// Mitsubishi GX Works2 project: PLC   PLC: FX3G
// LABEL_TEST

// global labels: Global1
VAR_GLOBAL
  MODBUS AT M50 : BOOL;  (* Modbus ON/OFF *)
  WeatherPrognose AT M30 : BOOL;  (* Waether prognose download *)
  Nordpool : BOOL;  (* Nordpool price *)
  Manual : BOOL;  (* Manual price *)
  UP_15_00 : BOOL;  (* Nordpool/naual data update *)
  Ready AT M1 : BOOL;  (* Machine ready *)
  NordPtoGeraph AT M64 : BOOL;  (* Nordpool Prise to graph *)
  CopyDataToGraph : BOOL;  (* Manual/Nordpool data copyng to graph *)
  CopyDataToGraphIsReady : BOOL;  (* Prise data is copyed to graph *)
  SortDataReady : BOOL;  (* Start sort data prodsedure ready *)
  EnergyUseGraph : BOOL;  (* Effective energy use next 24h *)
  DataLoading : BOOL;  (* Data Loading flag *)
  SortDataStart : BOOL;  (* Start data sorting *)
  SortData : BOOL;  (* Start sort data prodsedure *)
  MoveData : BOOL;  (* Move data to sort register *)
  SortDataOK : BOOL;  (* Data is sorted *)
  MoveDataOK : BOOL;  (* Data is moved *)
  Sort24hHighMinOK : BOOL;  (* Data is sorted *)
  Sort24hMinHighOK : BOOL;  (* Data sorted *)
  Sort24hMinHigh24OK : BOOL;  (* Data sorted *)
  Sort24hMinHigh : BOOL;  (* Sort 24h prise min to hight *)
  Sort24hHighMin : BOOL;  (* Sort 24h prise hight to min *)
  Sort24hMinHigh24 : BOOL;  (* Sort 24h prise Min to High *)
  price : BOOL;  (* Add nordpool manual pice *)
  FindPriseMax : BOOL;  (* Find max value in graph *)
  FindPriseMaxOK : BOOL;  (* Find max value is ready *)
  WeatherNextDay : BOOL;  (* Start weather next day prognisis calc *)
  NextDayAvrTemp AT D1850 : DINT;  (* Next day prognosis temp *)
  NextDayAvrWind AT D1852 : DINT;  (* Next day prognosis wind *)
  NextDayAvrCloudy AT D1854 : DINT;  (* Next day avareage cloudy prognosis *)
  WeatherNextDayOK : BOOL;  (* Weather next day OK *)
  ReadEnergyRequirement : BOOL;  (* Read energy requirement form enegry table *)
  ReadEnergyWind : INT;  (* wind prognosis information *)
  ReadEnergyRadiation : INT;  (* Enegri inoramatsion from prognaosis *)
  EnergyDataFromTable : INT;  (* energy information from the data table *)
  WriteEnergyRequirement : BOOL;  (* Write erengy requirements to data table *)
  WriteEnergyWind : INT;  (* Write energy to data table *)
  EnergyDataFromLast24h : INT;  (* Energy data from Last24H *)
  priceOK : BOOL;  (* Prse is selected *)
  GraphicDataUpdate : BOOL;  (* Update graphics data *)
  GraphicDataUpdateOK : BOOL;  (* Graphics data is updated *)
  SortDataGrReady : BOOL;  (* Data sorted for graphics *)
  EnernyUseReady : BOOL;  (* Egery graph is updated *)
  CalcUsablePriceThreshold : BOOL;  (* Calculate usable (low price) price threshold *)
  PorgnosGetButton AT M36 : BOOL;  (* Prognose Button HMI *)
  ReadEnergyRequirementOK : BOOL;  (* Read energy requirement is readed *)
  WriteEnergyRequirementOK : BOOL;  (* Write energy requirement is writed *)
  HeatFlowLiters AT D68 : INT;  (* Heat flow l/min *)
  Wifi_SSID AT D200 : ARRAY [0..31] OF INT;  (* WIfi SSID name *)
  RadiatorHeatingPump : BOOL;  (* Radiator Heat Pump ON/Off *)
  FloorHeatingPump : BOOL;  (* Floor heating pump ON/Off *)
  HeaterHeatingPump : BOOL;  (* Heter heating pump ON/Off *)
  ElectricHeaterCenter : BOOL;  (* Electric heater center positsion ON/OFF *)
  ElectricHeaterLower AT M14 : BOOL;  (* Electric heater lower ON/OFF *)
  RadiatorHeatingActuatorState : INT;  (* Radiator valve actuator positsion (0-100%hot) *)
  OutsideTemp AT D56 : INT;  (* Outside temp x10 *)
  Ring1TargetTemp AT D58 : DINT;  (* Ring 1 (Radiator) Target Temp *)
  Ring2TargetTemp AT D70 : INT;  (* Target temerature for floor heating *)
  RadiatorHeatTemp AT D36 : DINT;  (* Radiator heating temperatuse to heat *)
  Ring1ValvePos : INT;  (* Ring 1 Valve positsion *)
  FloorHeatTemp AT D40 : INT;  (* Floof heating temperatuse to heat *)
  FloorHeatingActuatorState : INT;  (* Floor heating positsion state (0..100% hot) *)
  HeatingMode : BOOL;  (* Heating or summer mode *)
  ElectricHeatON AT M40 : BOOL;  (* Electric heat method is ON *)
  SolidHeatON AT M41 : BOOL;  (* Solid fuel heteing method is ON *)
  HeatPumpHeatingON AT M42 : BOOL;  (* Heating pump heteing method is ON *)
  ElectricElementON : BOOL;  (* Switch electric heat ON *)
  PriceNow AT D2004 : INT;  (* Energy price now *)
  ElectricElementON_Sol_Heat : BOOL;  (* Heat element Solid Heat func *)
  ElectricElementON_El_Heat : BOOL;  (* Heat element ON Electric Heat func. *)
  TankWaterCapacity AT D2006 : INT;  (* Tenk water capasity *)
  TankEnergyCapacity100 AT D72 : DINT;  (* Tank Energy Capacity 100 *)
  EnergyConsumption24h AT D2008 : DINT;  (* Energy consumption last 24h *)
  HetedEnergyInLastH AT D2012 : INT;  (* Heting energy in last hours *)
  EnergyConsumptionYesterday AT D2010 : DINT;  (* Energy consumption yesterday *)
  ElElementPower AT D2014 : INT;  (* Heting element power W *)
  HeatingReallTime AT D2020 : DINT;  (* Real time heating (W) *)
  HeatingArea AT D1874 : DINT;  (* Heating area (building areme m2) *)
  PreviousDayWind : INT;  (* Previous day wind prognosis *)
  PreviousDayTemp : INT;  (* Previous day temperature probnosis *)
  PreviousDayCloudy : INT;  (* Previous day cloudy prognosis *)
  SolarRadiationDayMax : INT;  (* Solar radiation max per day *)
  EnConsumptionPer_C : DINT;  (* Energy consumption per degree *)
END_VAR

PROGRAM MAIN
VAR
  GraphicDataProtsess : INT;  (* Graphic data protsess count *)
END_VAR
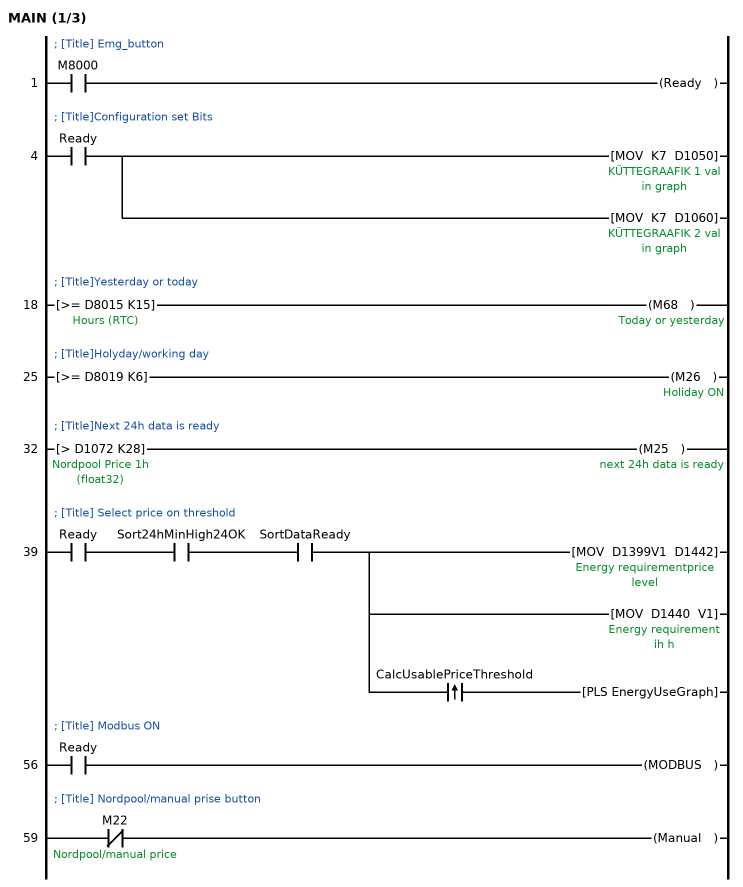
; [Title] Emg_button
1     LD      M8000
      OUT     Ready
; [Title]Configuration set Bits
4     LD      Ready
      MOV     K7 D1050  ; KÜTTEGRAAFIK 1 val in graph
        [note] 7 val. in heat cruve graph
      MOV     K7 D1060  ; KÜTTEGRAAFIK 2 val in graph
        [note] 7 val. in heat cruve graph
; [Title]Yesterday or today
18    LD>=    D8015 K15  ; Hours (RTC)
      OUT     M68  ; Today or yesterday
; [Title]Holyday/working day
25    LD>=    D8019 K6
      OUT     M26  ; Holiday ON
; [Title]Next 24h data is ready
32    LD>     D1072 K28  ; Nordpool Price 1h (float32)
      OUT     M25  ; next 24h data is ready
; [Title] Select price on threshold
39    LD      Ready
      AND     Sort24hMinHigh24OK
      AND     SortDataReady
      MOV     D1399V1 D1442  ; Energy requirementprice level
      MOV     D1440 V1  ; Energy requirement ih h
      ANDP    CalcUsablePriceThreshold
      PLS     EnergyUseGraph
; [Title] Modbus ON
56    LD      Ready
      OUT     MODBUS
; [Title] Nordpool/manual prise button
59    LDI     M22  ; Nordpool/manual price
      OUT     Manual
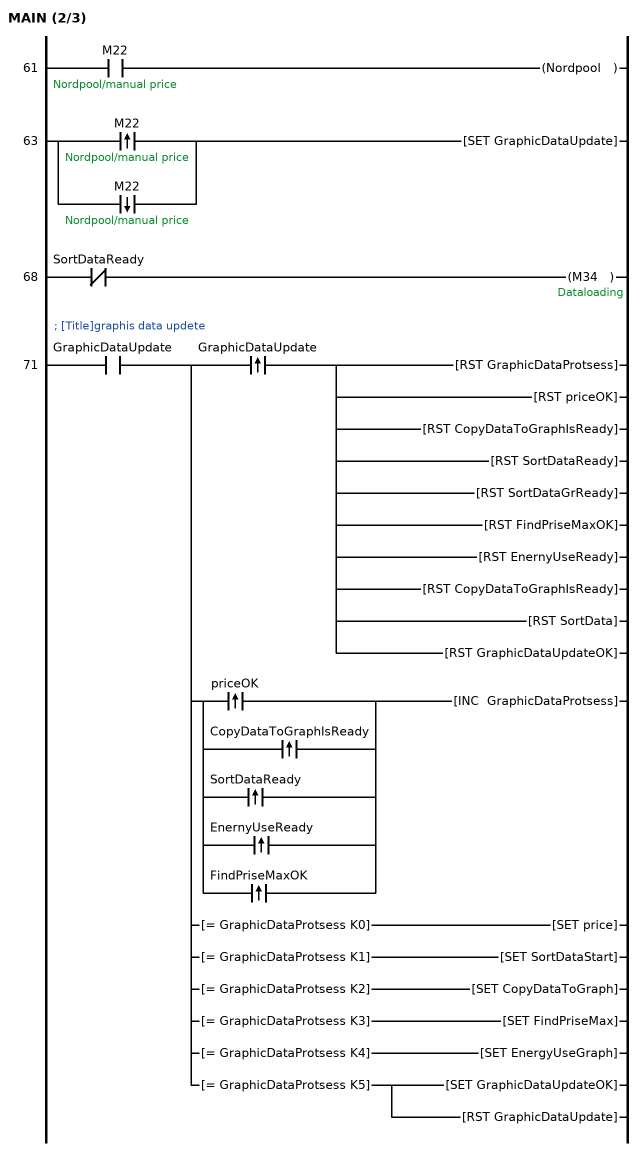
61    LD      M22  ; Nordpool/manual price
      OUT     Nordpool
63    LDP     M22  ; Nordpool/manual price
      ORF     M22  ; Nordpool/manual price
      SET     GraphicDataUpdate
68    LDI     SortDataReady
      OUT     M34  ; Dataloading
; [Title]graphis data updete
71    LD      GraphicDataUpdate
      MPS
      ANDP    GraphicDataUpdate
      RST     GraphicDataProtsess
      RST     priceOK
      RST     CopyDataToGraphIsReady
      RST     SortDataReady
      RST     SortDataGrReady
      RST     FindPriseMaxOK
      RST     EnernyUseReady
      RST     CopyDataToGraphIsReady
      RST     SortData
      RST     GraphicDataUpdateOK
      MRD
      LDP     priceOK
      ORP     CopyDataToGraphIsReady
      ORP     SortDataReady
      ORP     EnernyUseReady
      ORP     FindPriseMaxOK
      ANB
      INC     GraphicDataProtsess
      MRD
      AND=    GraphicDataProtsess K0
      SET     price
      MRD
      AND=    GraphicDataProtsess K1
      SET     SortDataStart
      MRD
      AND=    GraphicDataProtsess K2
      SET     CopyDataToGraph
      MRD
      AND=    GraphicDataProtsess K3
      SET     FindPriseMax
      MRD
      AND=    GraphicDataProtsess K4
      SET     EnergyUseGraph
      MPP
      AND=    GraphicDataProtsess K5
      SET     GraphicDataUpdateOK
      RST     GraphicDataUpdate
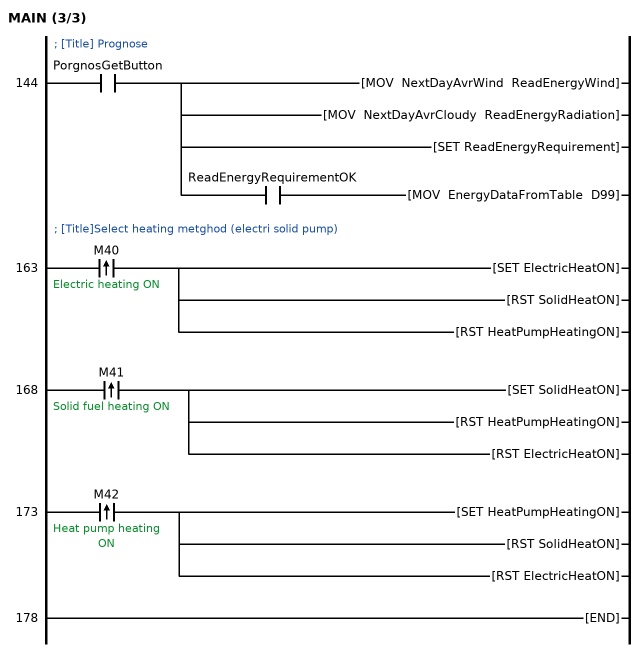
; [Title] Prognose
144   LD      PorgnosGetButton
      MOV     NextDayAvrWind ReadEnergyWind
      MOV     NextDayAvrCloudy ReadEnergyRadiation
      SET     ReadEnergyRequirement
      AND     ReadEnergyRequirementOK
      MOV     EnergyDataFromTable D99
; [Title]Select heating metghod (electri solid pump)
163   LDP     M40  ; Electric heating ON
      SET     ElectricHeatON
      RST     SolidHeatON
      RST     HeatPumpHeatingON
168   LDP     M41  ; Solid fuel heating ON
      SET     SolidHeatON
      RST     HeatPumpHeatingON
      RST     ElectricHeatON
173   LDP     M42  ; Heat pump heating ON
      SET     HeatPumpHeatingON
      RST     SolidHeatON
      RST     ElectricHeatON
178   END
END_PROGRAM

PROGRAM MODBUS
VAR
  ModBus_bnr : COUNTER;  (* Modbus comunicatsion block nr *)
  zxcv : BOOL;
END_VAR
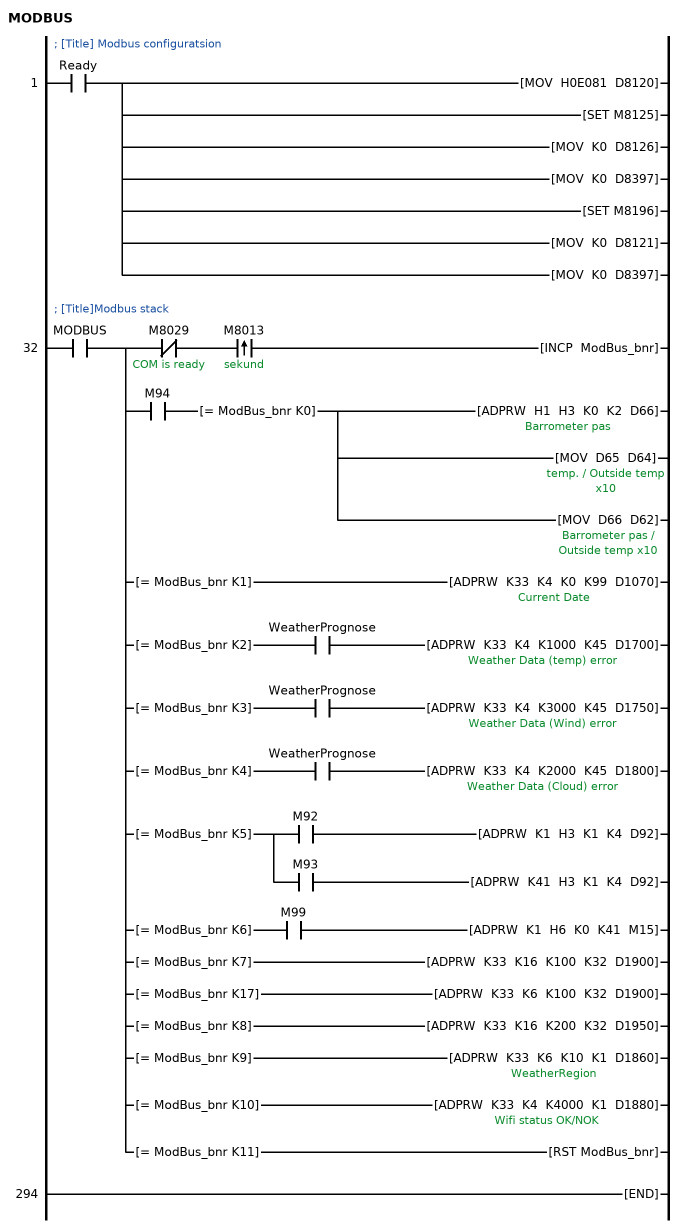
; [Title] Modbus configuratsion
1     LD      Ready
      MOV     H0E081 D8120
      SET     M8125
      MOV     K0 D8126
      MOV     K0 D8397
      SET     M8196
      MOV     K0 D8121
      MOV     K0 D8397
; [Title]Modbus stack
32    LD      MODBUS
      MPS
      ANI     M8029  ; COM is ready
      ANDP    M8013  ; sekund
      INCP    ModBus_bnr
        [note] barometer info
      MRD
      AND     M94
      AND=    ModBus_bnr K0
      ADPRW   H1 H3 K0 K2 D66  ; Barrometer pas
      MOV     D65 D64  ; temp. / Outside temp x10
      MOV     D66 D62  ; Outside temp x10
      MRD
      AND=    ModBus_bnr K1
      ADPRW   K33 K4 K0 K99 D1070  ; Current Date
        [note] Nordpool Data
      MRD
      AND=    ModBus_bnr K2
      AND     WeatherPrognose
      ADPRW   K33 K4 K1000 K45 D1700  ; Weather Data (temp) error
        [note] Weather Data (temp)
      MRD
      AND=    ModBus_bnr K3
      AND     WeatherPrognose
      ADPRW   K33 K4 K3000 K45 D1750  ; Weather Data (Wind) error
        [note] Weather Data (wind)
      MRD
      AND=    ModBus_bnr K4
      AND     WeatherPrognose
      ADPRW   K33 K4 K2000 K45 D1800  ; Weather Data (Cloud) error
        [note] Weather Data (cloudy%)
      MRD
      AND=    ModBus_bnr K5
      MPS
      AND     M92
      ADPRW   K1 H3 K1 K4 D92
        [note] Read pressure Data
      MPP
      AND     M93
      ADPRW   K41 H3 K1 K4 D92
        [note] Read pressure Data
      MRD
      AND=    ModBus_bnr K6
      AND     M99
      ADPRW   K1 H6 K0 K41 M15
        [note] PRESSURE SENSOR write MB 41
      MRD
      AND=    ModBus_bnr K7
      ADPRW   K33 K16 K100 K32 D1900
        [note] Wifi SSID
      MRD
      AND=    ModBus_bnr K17
      ADPRW   K33 K6 K100 K32 D1900
        [note] Wifi SSID
      MRD
      AND=    ModBus_bnr K8
      ADPRW   K33 K16 K200 K32 D1950
        [note] Wifi password
      MRD
      AND=    ModBus_bnr K9
      ADPRW   K33 K6 K10 K1 D1860  ; WeatherRegion
        [note] Weather region/loctsion
      MRD
      AND=    ModBus_bnr K10
      ADPRW   K33 K4 K4000 K1 D1880  ; Wifi status OK/NOK
        [note] Weather region/loctsion
      MPP
      AND=    ModBus_bnr K11
      RST     ModBus_bnr
294   END
END_PROGRAM

PROGRAM PRICE
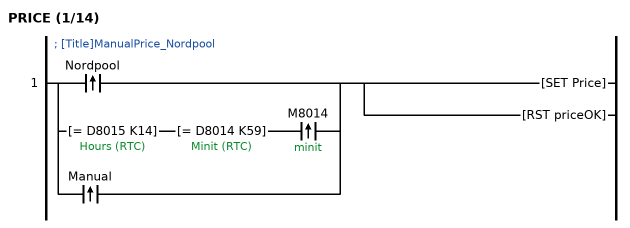
; [Title]ManualPrice_Nordpool
1     LDP     Nordpool
      LD=     D8015 K14  ; Hours (RTC)
      AND=    D8014 K59  ; Minit (RTC)
      ANDP    M8014  ; minit
      ORB
      ORP     Manual
      SET     Price
      RST     priceOK
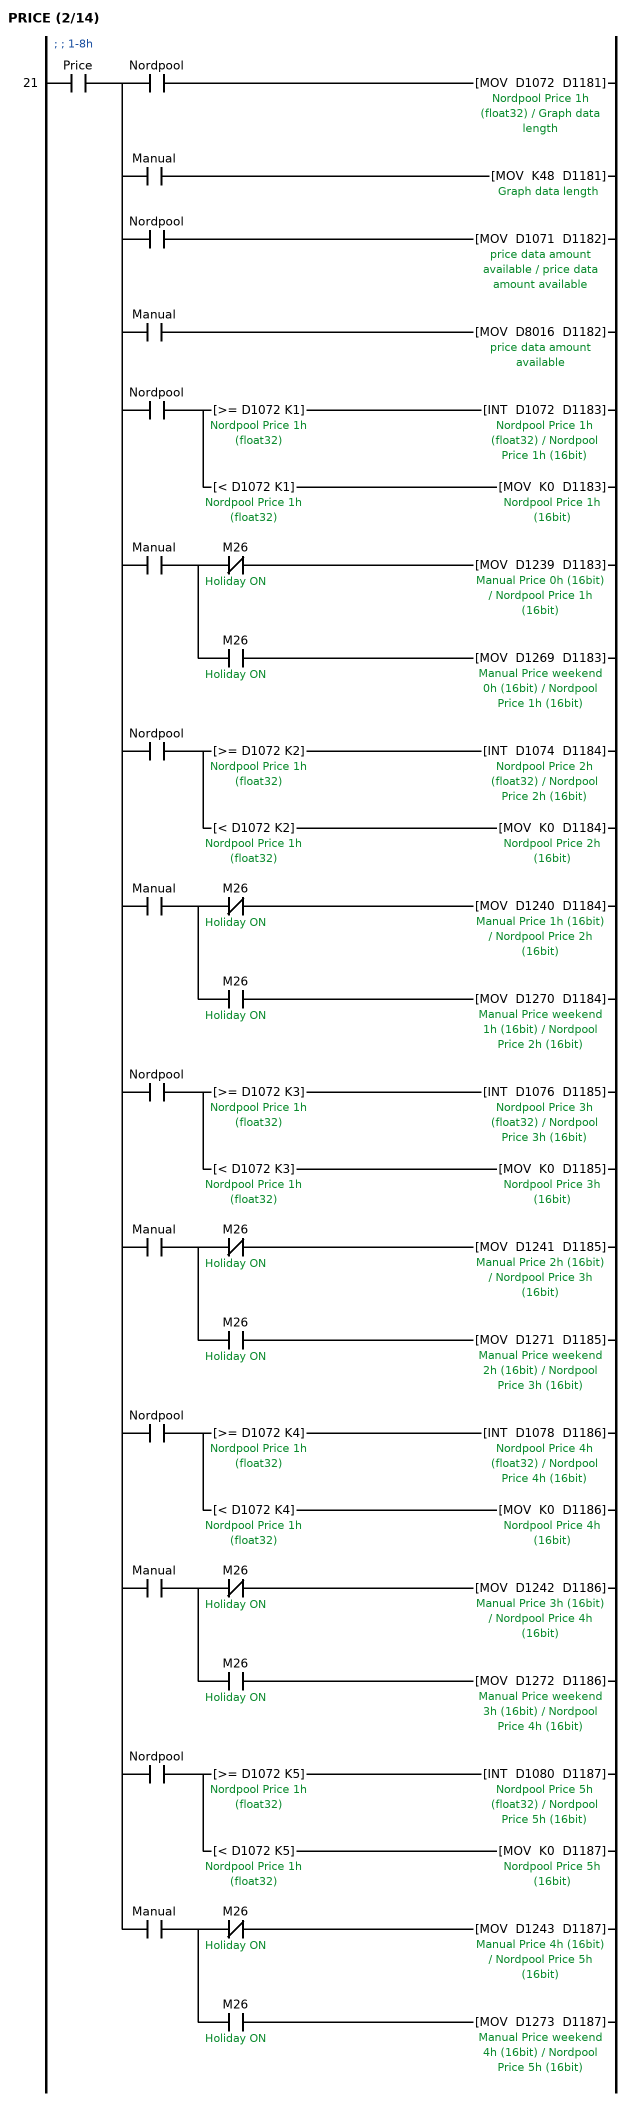
;  1-8h
21    LD      Price
      MPS
      AND     Nordpool
      MOV     D1072 D1181  ; Nordpool Price 1h (float32) / Graph data length
        [note] 00-01
      MRD
      AND     Manual
      MOV     K48 D1181
      MRD
      AND     Nordpool
      MOV     D1071 D1182  ; price data amount available / price data amount available
      MRD
      AND     Manual
      MOV     D8016 D1182
      MRD
      AND     Nordpool
      MPS
      AND>=   D1072 K1  ; Nordpool Price 1h (float32)
      INT     D1072 D1183  ; Nordpool Price 1h (16bit)
      MPP
      AND<    D1072 K1  ; Nordpool Price 1h (float32)
      MOV     K0 D1183
      MRD
      AND     Manual
      MPS
      ANI     M26  ; Holiday ON
      MOV     D1239 D1183  ; Manual Price 0h (16bit)
      MPP
      AND     M26  ; Holiday ON
      MOV     D1269 D1183  ; Manual Price weekend 0h (16bit)
      MRD
      AND     Nordpool
      MPS
      AND>=   D1072 K2  ; Nordpool Price 1h (float32)
      INT     D1074 D1184  ; Nordpool Price 2h (float32) / Nordpool Price 2h (16bit)
        [note] 01-02
      MPP
      AND<    D1072 K2  ; Nordpool Price 1h (float32)
      MOV     K0 D1184
      MRD
      AND     Manual
      MPS
      ANI     M26  ; Holiday ON
      MOV     D1240 D1184  ; Manual Price 1h (16bit)
      MPP
      AND     M26  ; Holiday ON
      MOV     D1270 D1184  ; Manual Price weekend 1h (16bit)
      MRD
      AND     Nordpool
      MPS
      AND>=   D1072 K3  ; Nordpool Price 1h (float32)
      INT     D1076 D1185  ; Nordpool Price 3h (float32) / Nordpool Price 3h (16bit)
        [note] 02-03
      MPP
      AND<    D1072 K3  ; Nordpool Price 1h (float32)
      MOV     K0 D1185
      MRD
      AND     Manual
      MPS
      ANI     M26  ; Holiday ON
      MOV     D1241 D1185  ; Manual Price 2h (16bit)
      MPP
      AND     M26  ; Holiday ON
      MOV     D1271 D1185  ; Manual Price weekend 2h (16bit)
      MRD
      AND     Nordpool
      MPS
      AND>=   D1072 K4  ; Nordpool Price 1h (float32)
      INT     D1078 D1186  ; Nordpool Price 4h (float32) / Nordpool Price 4h (16bit)
        [note] 03-04
      MPP
      AND<    D1072 K4  ; Nordpool Price 1h (float32)
      MOV     K0 D1186
      MRD
      AND     Manual
      MPS
      ANI     M26  ; Holiday ON
      MOV     D1242 D1186  ; Manual Price 3h (16bit)
      MPP
      AND     M26  ; Holiday ON
      MOV     D1272 D1186  ; Manual Price weekend 3h (16bit)
      MRD
      AND     Nordpool
      MPS
      AND>=   D1072 K5  ; Nordpool Price 1h (float32)
      INT     D1080 D1187  ; Nordpool Price 5h (float32) / Nordpool Price 5h (16bit)
        [note] 04-05
      MPP
      AND<    D1072 K5  ; Nordpool Price 1h (float32)
      MOV     K0 D1187
      MPP
      AND     Manual
      MPS
      ANI     M26  ; Holiday ON
      MOV     D1243 D1187  ; Manual Price 4h (16bit)
      MPP
      AND     M26  ; Holiday ON
      MOV     D1273 D1187  ; Manual Price weekend 4h (16bit)
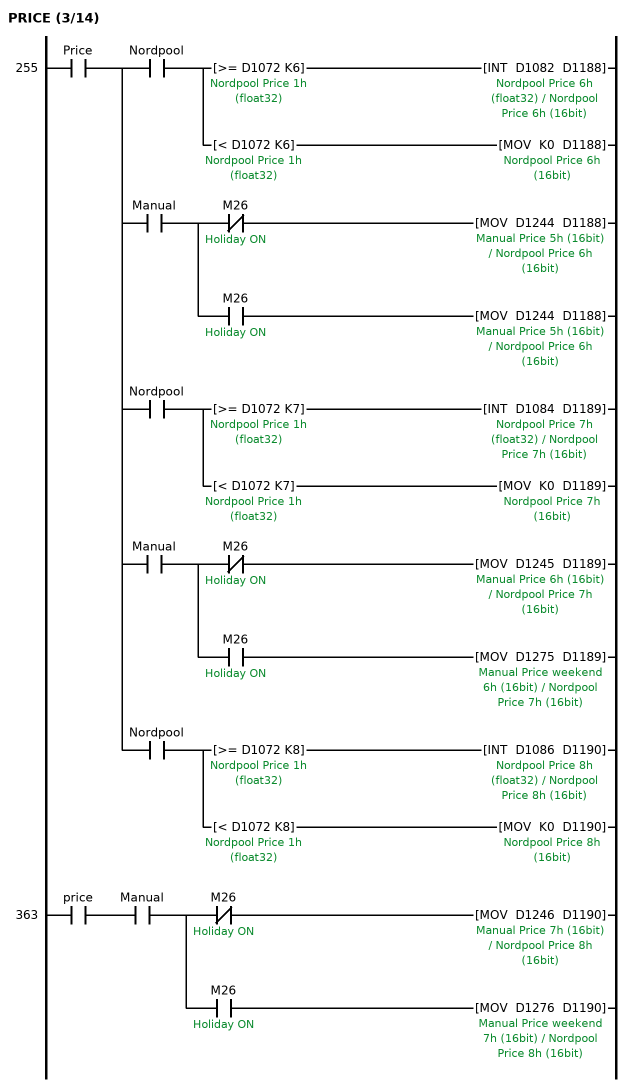
255   LD      Price
      MPS
      AND     Nordpool
      MPS
      AND>=   D1072 K6  ; Nordpool Price 1h (float32)
      INT     D1082 D1188  ; Nordpool Price 6h (float32) / Nordpool Price 6h (16bit)
        [note] 05-06
      MPP
      AND<    D1072 K6  ; Nordpool Price 1h (float32)
      MOV     K0 D1188
      MRD
      AND     Manual
      MPS
      ANI     M26  ; Holiday ON
      MOV     D1244 D1188  ; Manual Price 5h (16bit)
      MPP
      AND     M26  ; Holiday ON
      MOV     D1244 D1188
      MRD
      AND     Nordpool
      MPS
      AND>=   D1072 K7  ; Nordpool Price 1h (float32)
      INT     D1084 D1189  ; Nordpool Price 7h (float32) / Nordpool Price 7h (16bit)
        [note] 06-07
      MPP
      AND<    D1072 K7  ; Nordpool Price 1h (float32)
      MOV     K0 D1189
      MRD
      AND     Manual
      MPS
      ANI     M26  ; Holiday ON
      MOV     D1245 D1189  ; Manual Price 6h (16bit)
      MPP
      AND     M26  ; Holiday ON
      MOV     D1275 D1189  ; Manual Price weekend 6h (16bit)
      MPP
      AND     Nordpool
      MPS
      AND>=   D1072 K8  ; Nordpool Price 1h (float32)
      INT     D1086 D1190  ; Nordpool Price 8h (float32) / Nordpool Price 8h (16bit)
        [note] 07-08
      MPP
      AND<    D1072 K8  ; Nordpool Price 1h (float32)
      MOV     K0 D1190
363   LD      price
      AND     Manual
      MPS
      ANI     M26  ; Holiday ON
      MOV     D1246 D1190  ; Manual Price 7h (16bit)
      MPP
      AND     M26  ; Holiday ON
      MOV     D1276 D1190  ; Manual Price weekend 7h (16bit)
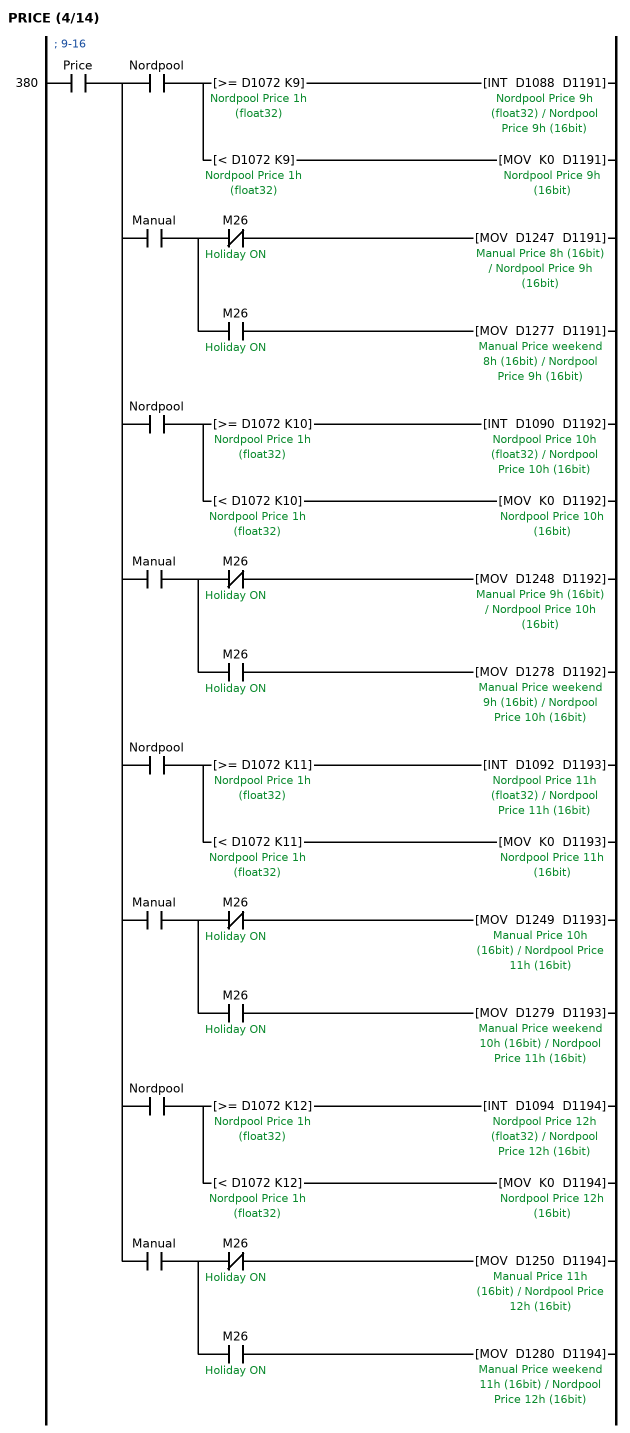
; 9-16
380   LD      Price
      MPS
      AND     Nordpool
      MPS
      AND>=   D1072 K9  ; Nordpool Price 1h (float32)
      INT     D1088 D1191  ; Nordpool Price 9h (float32) / Nordpool Price 9h (16bit)
        [note] 08-09
      MPP
      AND<    D1072 K9  ; Nordpool Price 1h (float32)
      MOV     K0 D1191
      MRD
      AND     Manual
      MPS
      ANI     M26  ; Holiday ON
      MOV     D1247 D1191  ; Manual Price 8h (16bit)
      MPP
      AND     M26  ; Holiday ON
      MOV     D1277 D1191  ; Manual Price weekend 8h (16bit)
      MRD
      AND     Nordpool
      MPS
      AND>=   D1072 K10  ; Nordpool Price 1h (float32)
      INT     D1090 D1192  ; Nordpool Price 10h (float32) / Nordpool Price 10h (16bit)
        [note] 9-10
      MPP
      AND<    D1072 K10  ; Nordpool Price 1h (float32)
      MOV     K0 D1192
      MRD
      AND     Manual
      MPS
      ANI     M26  ; Holiday ON
      MOV     D1248 D1192  ; Manual Price 9h (16bit)
      MPP
      AND     M26  ; Holiday ON
      MOV     D1278 D1192  ; Manual Price weekend 9h (16bit)
      MRD
      AND     Nordpool
      MPS
      AND>=   D1072 K11  ; Nordpool Price 1h (float32)
      INT     D1092 D1193  ; Nordpool Price 11h (float32) / Nordpool Price 11h (16bit)
        [note] 10-11
      MPP
      AND<    D1072 K11  ; Nordpool Price 1h (float32)
      MOV     K0 D1193
      MRD
      AND     Manual
      MPS
      ANI     M26  ; Holiday ON
      MOV     D1249 D1193  ; Manual Price 10h (16bit)
      MPP
      AND     M26  ; Holiday ON
      MOV     D1279 D1193  ; Manual Price weekend 10h (16bit)
      MRD
      AND     Nordpool
      MPS
      AND>=   D1072 K12  ; Nordpool Price 1h (float32)
      INT     D1094 D1194  ; Nordpool Price 12h (float32) / Nordpool Price 12h (16bit)
        [note] 11-12
      MPP
      AND<    D1072 K12  ; Nordpool Price 1h (float32)
      MOV     K0 D1194
      MPP
      AND     Manual
      MPS
      ANI     M26  ; Holiday ON
      MOV     D1250 D1194  ; Manual Price 11h (16bit)
      MPP
      AND     M26  ; Holiday ON
      MOV     D1280 D1194  ; Manual Price weekend 11h (16bit)
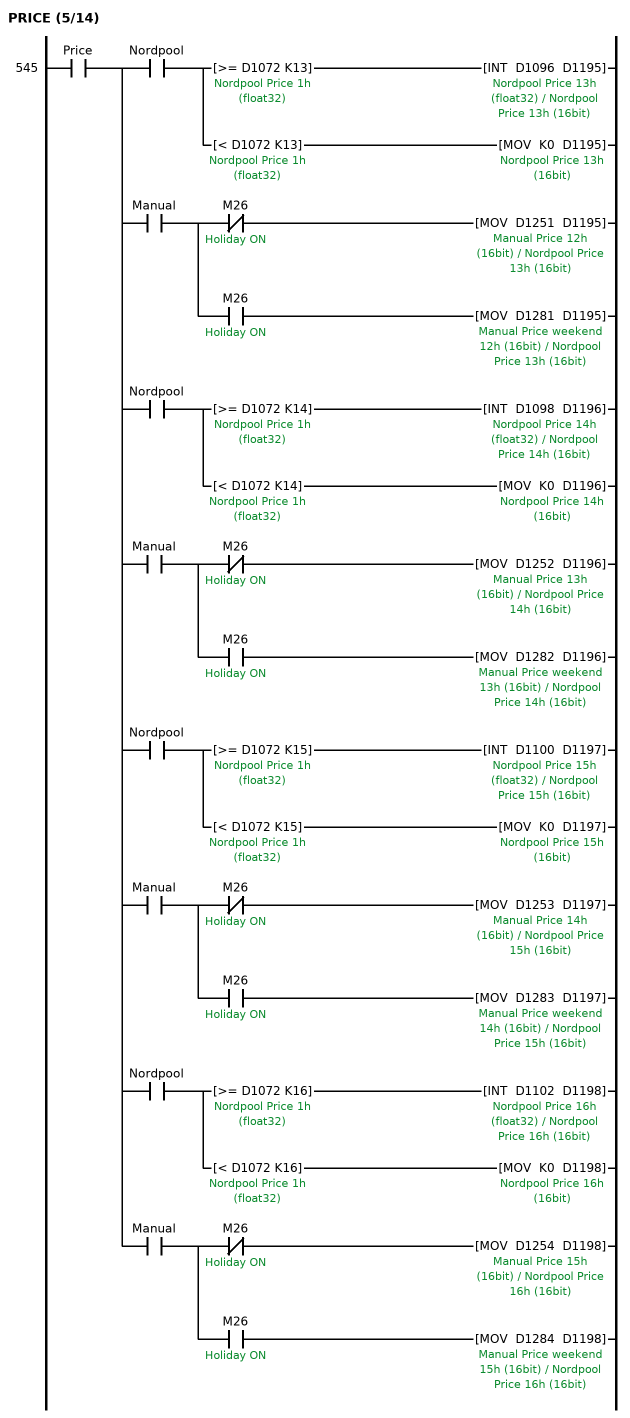
545   LD      Price
      MPS
      AND     Nordpool
      MPS
      AND>=   D1072 K13  ; Nordpool Price 1h (float32)
      INT     D1096 D1195  ; Nordpool Price 13h (float32) / Nordpool Price 13h (16bit)
        [note] 12-13
      MPP
      AND<    D1072 K13  ; Nordpool Price 1h (float32)
      MOV     K0 D1195
      MRD
      AND     Manual
      MPS
      ANI     M26  ; Holiday ON
      MOV     D1251 D1195  ; Manual Price 12h (16bit)
      MPP
      AND     M26  ; Holiday ON
      MOV     D1281 D1195  ; Manual Price weekend 12h (16bit)
      MRD
      AND     Nordpool
      MPS
      AND>=   D1072 K14  ; Nordpool Price 1h (float32)
      INT     D1098 D1196  ; Nordpool Price 14h (float32) / Nordpool Price 14h (16bit)
        [note] 13-14
      MPP
      AND<    D1072 K14  ; Nordpool Price 1h (float32)
      MOV     K0 D1196
      MRD
      AND     Manual
      MPS
      ANI     M26  ; Holiday ON
      MOV     D1252 D1196  ; Manual Price 13h (16bit)
      MPP
      AND     M26  ; Holiday ON
      MOV     D1282 D1196  ; Manual Price weekend 13h (16bit)
      MRD
      AND     Nordpool
      MPS
      AND>=   D1072 K15  ; Nordpool Price 1h (float32)
      INT     D1100 D1197  ; Nordpool Price 15h (float32) / Nordpool Price 15h (16bit)
        [note] 14-15
      MPP
      AND<    D1072 K15  ; Nordpool Price 1h (float32)
      MOV     K0 D1197
      MRD
      AND     Manual
      MPS
      ANI     M26  ; Holiday ON
      MOV     D1253 D1197  ; Manual Price 14h (16bit)
      MPP
      AND     M26  ; Holiday ON
      MOV     D1283 D1197  ; Manual Price weekend 14h (16bit)
      MRD
      AND     Nordpool
      MPS
      AND>=   D1072 K16  ; Nordpool Price 1h (float32)
      INT     D1102 D1198  ; Nordpool Price 16h (float32) / Nordpool Price 16h (16bit)
        [note] 15-16
      MPP
      AND<    D1072 K16  ; Nordpool Price 1h (float32)
      MOV     K0 D1198
      MPP
      AND     Manual
      MPS
      ANI     M26  ; Holiday ON
      MOV     D1254 D1198  ; Manual Price 15h (16bit)
      MPP
      AND     M26  ; Holiday ON
      MOV     D1284 D1198  ; Manual Price weekend 15h (16bit)
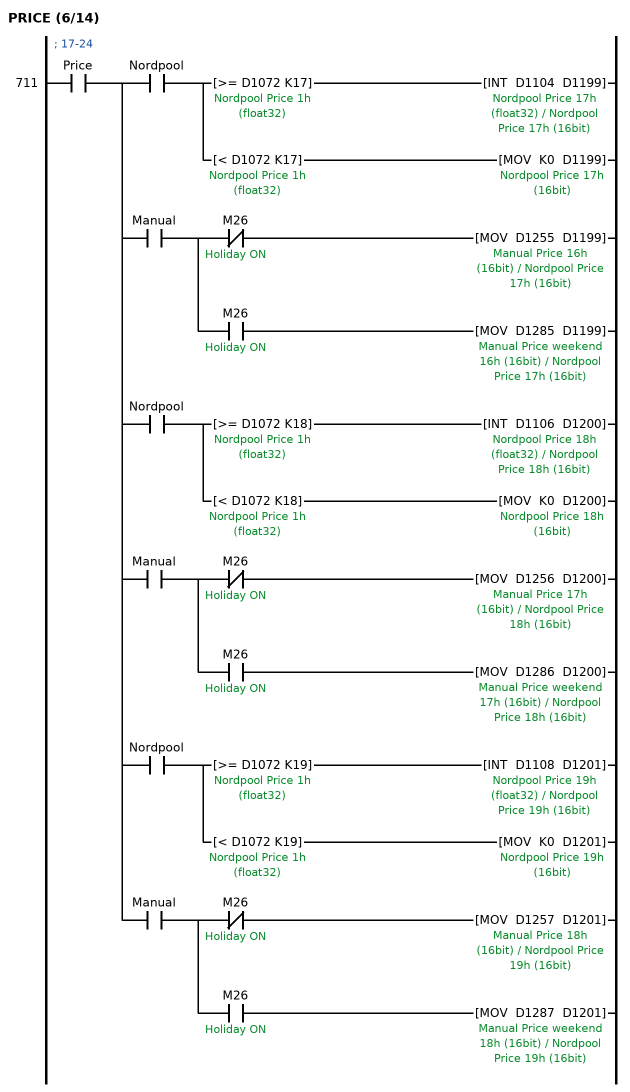
; 17-24
711   LD      Price
      MPS
      AND     Nordpool
      MPS
      AND>=   D1072 K17  ; Nordpool Price 1h (float32)
      INT     D1104 D1199  ; Nordpool Price 17h (float32) / Nordpool Price 17h (16bit)
        [note] 16-17
      MPP
      AND<    D1072 K17  ; Nordpool Price 1h (float32)
      MOV     K0 D1199
      MRD
      AND     Manual
      MPS
      ANI     M26  ; Holiday ON
      MOV     D1255 D1199  ; Manual Price 16h (16bit)
      MPP
      AND     M26  ; Holiday ON
      MOV     D1285 D1199  ; Manual Price weekend 16h (16bit)
      MRD
      AND     Nordpool
      MPS
      AND>=   D1072 K18  ; Nordpool Price 1h (float32)
      INT     D1106 D1200  ; Nordpool Price 18h (float32) / Nordpool Price 18h (16bit)
        [note] 17-18
      MPP
      AND<    D1072 K18  ; Nordpool Price 1h (float32)
      MOV     K0 D1200
      MRD
      AND     Manual
      MPS
      ANI     M26  ; Holiday ON
      MOV     D1256 D1200  ; Manual Price 17h (16bit)
      MPP
      AND     M26  ; Holiday ON
      MOV     D1286 D1200  ; Manual Price weekend 17h (16bit)
      MRD
      AND     Nordpool
      MPS
      AND>=   D1072 K19  ; Nordpool Price 1h (float32)
      INT     D1108 D1201  ; Nordpool Price 19h (float32) / Nordpool Price 19h (16bit)
        [note] 18-19
      MPP
      AND<    D1072 K19  ; Nordpool Price 1h (float32)
      MOV     K0 D1201
      MPP
      AND     Manual
      MPS
      ANI     M26  ; Holiday ON
      MOV     D1257 D1201  ; Manual Price 18h (16bit)
      MPP
      AND     M26  ; Holiday ON
      MOV     D1287 D1201  ; Manual Price weekend 18h (16bit)
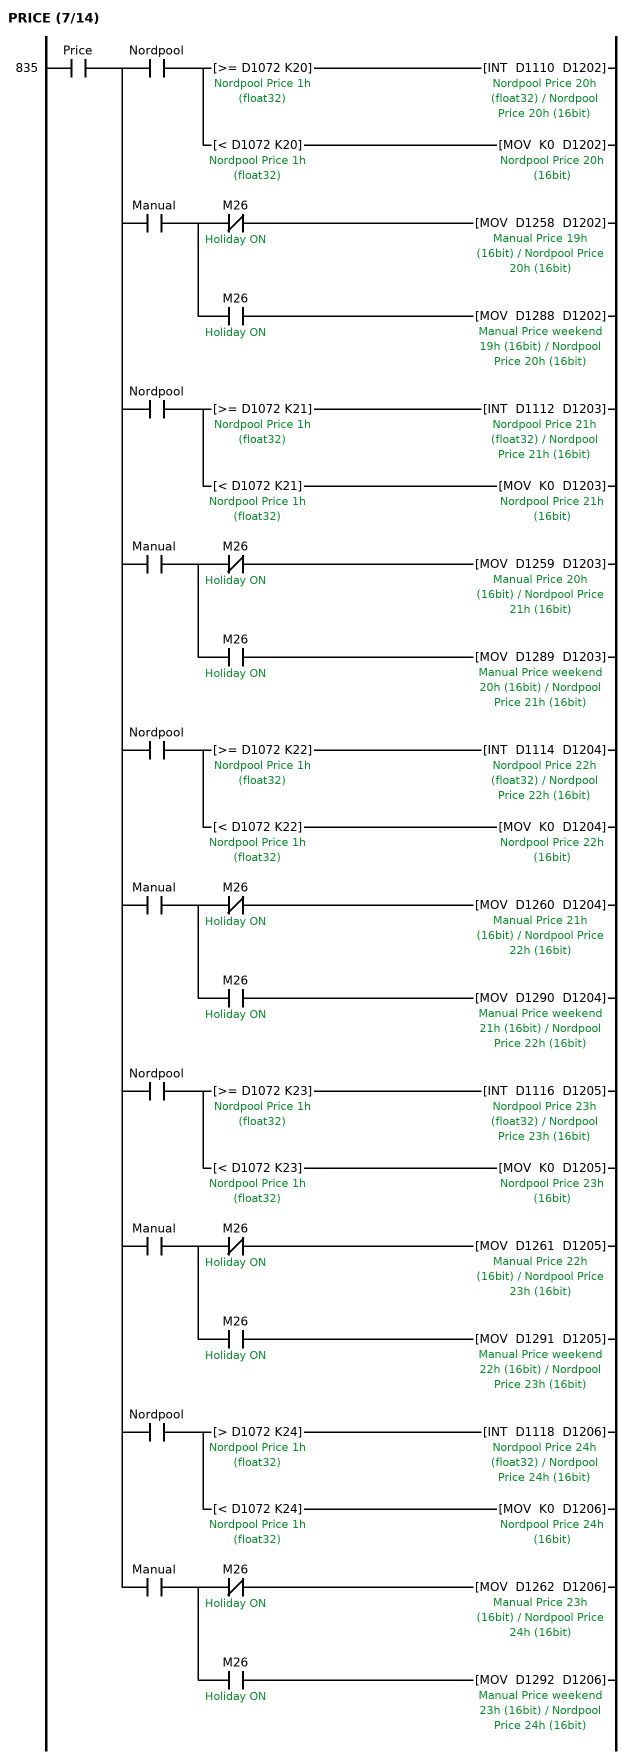
835   LD      Price
      MPS
      AND     Nordpool
      MPS
      AND>=   D1072 K20  ; Nordpool Price 1h (float32)
      INT     D1110 D1202  ; Nordpool Price 20h (float32) / Nordpool Price 20h (16bit)
        [note] 19-20
      MPP
      AND<    D1072 K20  ; Nordpool Price 1h (float32)
      MOV     K0 D1202
      MRD
      AND     Manual
      MPS
      ANI     M26  ; Holiday ON
      MOV     D1258 D1202  ; Manual Price 19h (16bit)
      MPP
      AND     M26  ; Holiday ON
      MOV     D1288 D1202  ; Manual Price weekend 19h (16bit)
      MRD
      AND     Nordpool
      MPS
      AND>=   D1072 K21  ; Nordpool Price 1h (float32)
      INT     D1112 D1203  ; Nordpool Price 21h (float32) / Nordpool Price 21h (16bit)
        [note] 20-21
      MPP
      AND<    D1072 K21  ; Nordpool Price 1h (float32)
      MOV     K0 D1203
      MRD
      AND     Manual
      MPS
      ANI     M26  ; Holiday ON
      MOV     D1259 D1203  ; Manual Price 20h (16bit)
      MPP
      AND     M26  ; Holiday ON
      MOV     D1289 D1203  ; Manual Price weekend 20h (16bit)
      MRD
      AND     Nordpool
      MPS
      AND>=   D1072 K22  ; Nordpool Price 1h (float32)
      INT     D1114 D1204  ; Nordpool Price 22h (float32) / Nordpool Price 22h (16bit)
        [note] 21-22
      MPP
      AND<    D1072 K22  ; Nordpool Price 1h (float32)
      MOV     K0 D1204
      MRD
      AND     Manual
      MPS
      ANI     M26  ; Holiday ON
      MOV     D1260 D1204  ; Manual Price 21h (16bit)
      MPP
      AND     M26  ; Holiday ON
      MOV     D1290 D1204  ; Manual Price weekend 21h (16bit)
      MRD
      AND     Nordpool
      MPS
      AND>=   D1072 K23  ; Nordpool Price 1h (float32)
      INT     D1116 D1205  ; Nordpool Price 23h (float32) / Nordpool Price 23h (16bit)
        [note] 22-23
      MPP
      AND<    D1072 K23  ; Nordpool Price 1h (float32)
      MOV     K0 D1205
      MRD
      AND     Manual
      MPS
      ANI     M26  ; Holiday ON
      MOV     D1261 D1205  ; Manual Price 22h (16bit)
      MPP
      AND     M26  ; Holiday ON
      MOV     D1291 D1205  ; Manual Price weekend 22h (16bit)
      MRD
      AND     Nordpool
      MPS
      AND>    D1072 K24  ; Nordpool Price 1h (float32)
      INT     D1118 D1206  ; Nordpool Price 24h (float32) / Nordpool Price 24h (16bit)
        [note] 23-00
      MPP
      AND<    D1072 K24  ; Nordpool Price 1h (float32)
      MOV     K0 D1206
      MPP
      AND     Manual
      MPS
      ANI     M26  ; Holiday ON
      MOV     D1262 D1206  ; Manual Price 23h (16bit)
      MPP
      AND     M26  ; Holiday ON
      MOV     D1292 D1206  ; Manual Price weekend 23h (16bit)
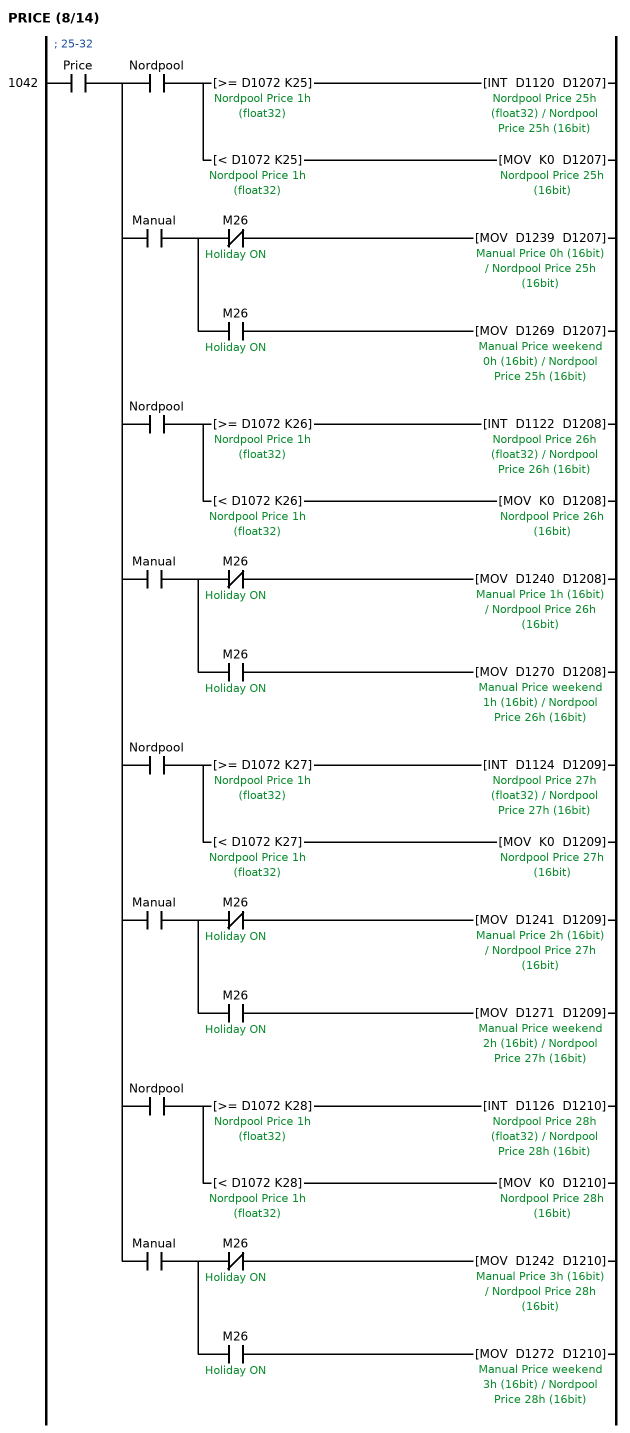
; 25-32
1042  LD      Price
      MPS
      AND     Nordpool
      MPS
      AND>=   D1072 K25  ; Nordpool Price 1h (float32)
      INT     D1120 D1207  ; Nordpool Price 25h (float32) / Nordpool Price 25h (16bit)
        [note] 25-26 (00-01)
      MPP
      AND<    D1072 K25  ; Nordpool Price 1h (float32)
      MOV     K0 D1207
      MRD
      AND     Manual
      MPS
      ANI     M26  ; Holiday ON
      MOV     D1239 D1207
      MPP
      AND     M26  ; Holiday ON
      MOV     D1269 D1207
      MRD
      AND     Nordpool
      MPS
      AND>=   D1072 K26  ; Nordpool Price 1h (float32)
      INT     D1122 D1208  ; Nordpool Price 26h (float32) / Nordpool Price 26h (16bit)
        [note] 26-27 (01-02)
      MPP
      AND<    D1072 K26  ; Nordpool Price 1h (float32)
      MOV     K0 D1208
      MRD
      AND     Manual
      MPS
      ANI     M26  ; Holiday ON
      MOV     D1240 D1208
      MPP
      AND     M26  ; Holiday ON
      MOV     D1270 D1208
      MRD
      AND     Nordpool
      MPS
      AND>=   D1072 K27  ; Nordpool Price 1h (float32)
      INT     D1124 D1209  ; Nordpool Price 27h (float32) / Nordpool Price 27h (16bit)
        [note] 27-28 (02-03)
      MPP
      AND<    D1072 K27  ; Nordpool Price 1h (float32)
      MOV     K0 D1209
      MRD
      AND     Manual
      MPS
      ANI     M26  ; Holiday ON
      MOV     D1241 D1209
      MPP
      AND     M26  ; Holiday ON
      MOV     D1271 D1209
      MRD
      AND     Nordpool
      MPS
      AND>=   D1072 K28  ; Nordpool Price 1h (float32)
      INT     D1126 D1210  ; Nordpool Price 28h (float32) / Nordpool Price 28h (16bit)
        [note] 28-29 (03-04)
      MPP
      AND<    D1072 K28  ; Nordpool Price 1h (float32)
      MOV     K0 D1210
      MPP
      AND     Manual
      MPS
      ANI     M26  ; Holiday ON
      MOV     D1242 D1210
      MPP
      AND     M26  ; Holiday ON
      MOV     D1272 D1210
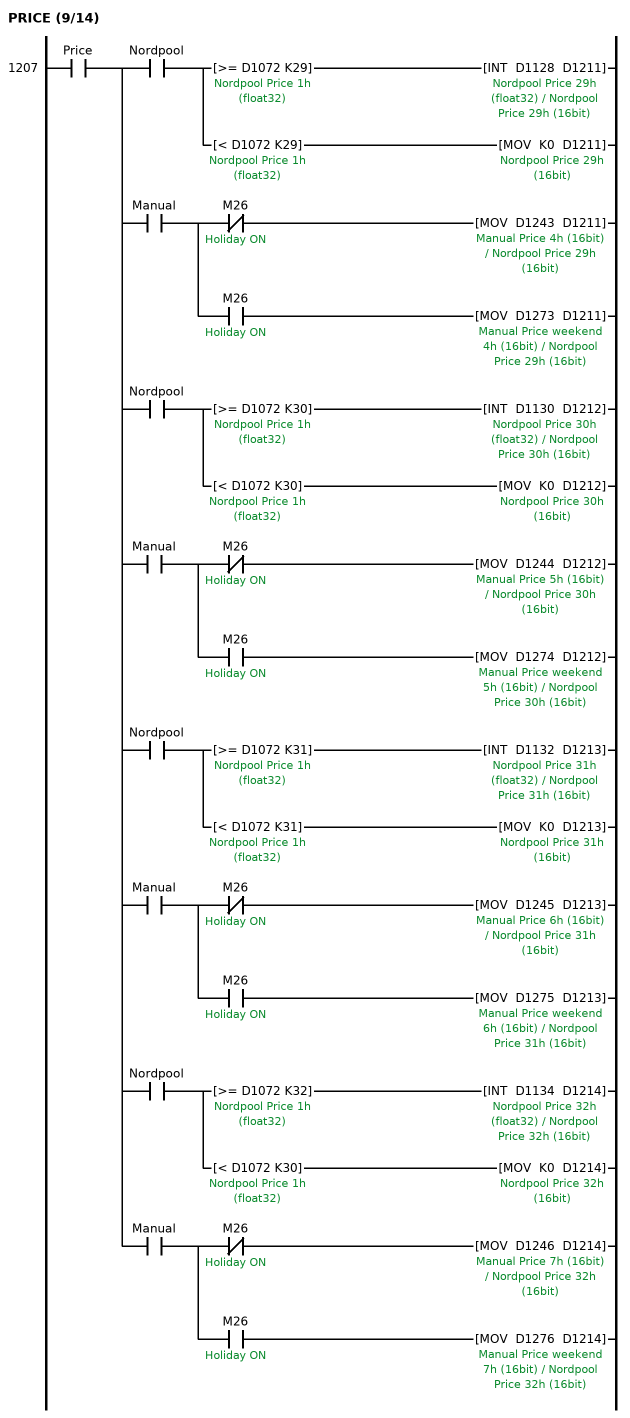
1207  LD      Price
      MPS
      AND     Nordpool
      MPS
      AND>=   D1072 K29  ; Nordpool Price 1h (float32)
      INT     D1128 D1211  ; Nordpool Price 29h (float32) / Nordpool Price 29h (16bit)
        [note] 29-30 (04-05)
      MPP
      AND<    D1072 K29  ; Nordpool Price 1h (float32)
      MOV     K0 D1211
      MRD
      AND     Manual
      MPS
      ANI     M26  ; Holiday ON
      MOV     D1243 D1211
      MPP
      AND     M26  ; Holiday ON
      MOV     D1273 D1211
      MRD
      AND     Nordpool
      MPS
      AND>=   D1072 K30  ; Nordpool Price 1h (float32)
      INT     D1130 D1212  ; Nordpool Price 30h (float32) / Nordpool Price 30h (16bit)
        [note] ; 30-31 (05-06)
      MPP
      AND<    D1072 K30  ; Nordpool Price 1h (float32)
      MOV     K0 D1212
      MRD
      AND     Manual
      MPS
      ANI     M26  ; Holiday ON
      MOV     D1244 D1212
      MPP
      AND     M26  ; Holiday ON
      MOV     D1274 D1212  ; Manual Price weekend 5h (16bit)
      MRD
      AND     Nordpool
      MPS
      AND>=   D1072 K31  ; Nordpool Price 1h (float32)
      INT     D1132 D1213  ; Nordpool Price 31h (float32) / Nordpool Price 31h (16bit)
        [note] 31-32 (06-07)
      MPP
      AND<    D1072 K31  ; Nordpool Price 1h (float32)
      MOV     K0 D1213
      MRD
      AND     Manual
      MPS
      ANI     M26  ; Holiday ON
      MOV     D1245 D1213
      MPP
      AND     M26  ; Holiday ON
      MOV     D1275 D1213
      MRD
      AND     Nordpool
      MPS
      AND>=   D1072 K32  ; Nordpool Price 1h (float32)
      INT     D1134 D1214  ; Nordpool Price 32h (float32) / Nordpool Price 32h (16bit)
        [note] 32-33 (07-08)
      MPP
      AND<    D1072 K30  ; Nordpool Price 1h (float32)
      MOV     K0 D1214
      MPP
      AND     Manual
      MPS
      ANI     M26  ; Holiday ON
      MOV     D1246 D1214
      MPP
      AND     M26  ; Holiday ON
      MOV     D1276 D1214
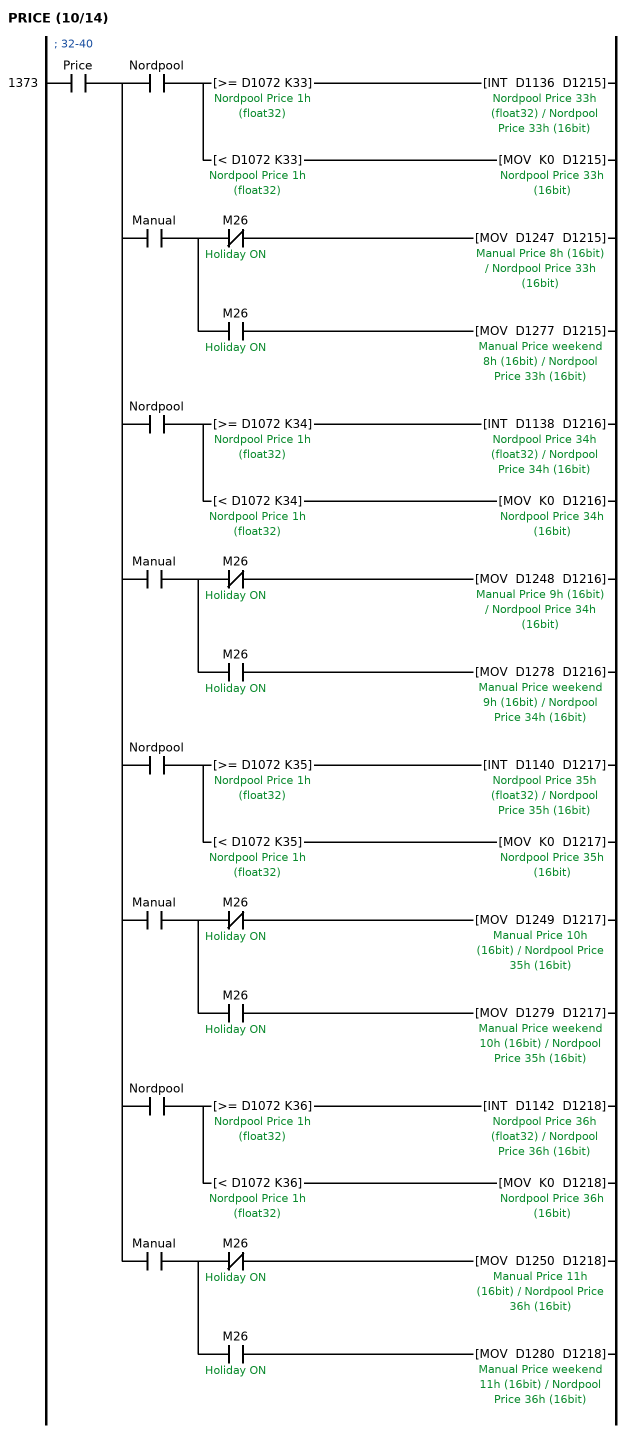
; 32-40
1373  LD      Price
      MPS
      AND     Nordpool
      MPS
      AND>=   D1072 K33  ; Nordpool Price 1h (float32)
      INT     D1136 D1215  ; Nordpool Price 33h (float32) / Nordpool Price 33h (16bit)
        [note] ;33-34 (08-09)
      MPP
      AND<    D1072 K33  ; Nordpool Price 1h (float32)
      MOV     K0 D1215
      MRD
      AND     Manual
      MPS
      ANI     M26  ; Holiday ON
      MOV     D1247 D1215
      MPP
      AND     M26  ; Holiday ON
      MOV     D1277 D1215
      MRD
      AND     Nordpool
      MPS
      AND>=   D1072 K34  ; Nordpool Price 1h (float32)
      INT     D1138 D1216  ; Nordpool Price 34h (float32) / Nordpool Price 34h (16bit)
        [note] 34-35 (09-10)
      MPP
      AND<    D1072 K34  ; Nordpool Price 1h (float32)
      MOV     K0 D1216
      MRD
      AND     Manual
      MPS
      ANI     M26  ; Holiday ON
      MOV     D1248 D1216
      MPP
      AND     M26  ; Holiday ON
      MOV     D1278 D1216
      MRD
      AND     Nordpool
      MPS
      AND>=   D1072 K35  ; Nordpool Price 1h (float32)
      INT     D1140 D1217  ; Nordpool Price 35h (float32) / Nordpool Price 35h (16bit)
        [note] 35-36 (10-11)
      MPP
      AND<    D1072 K35  ; Nordpool Price 1h (float32)
      MOV     K0 D1217
      MRD
      AND     Manual
      MPS
      ANI     M26  ; Holiday ON
      MOV     D1249 D1217
      MPP
      AND     M26  ; Holiday ON
      MOV     D1279 D1217
      MRD
      AND     Nordpool
      MPS
      AND>=   D1072 K36  ; Nordpool Price 1h (float32)
      INT     D1142 D1218  ; Nordpool Price 36h (float32) / Nordpool Price 36h (16bit)
        [note] 36-37 (11-12)
      MPP
      AND<    D1072 K36  ; Nordpool Price 1h (float32)
      MOV     K0 D1218
      MPP
      AND     Manual
      MPS
      ANI     M26  ; Holiday ON
      MOV     D1250 D1218
      MPP
      AND     M26  ; Holiday ON
      MOV     D1280 D1218
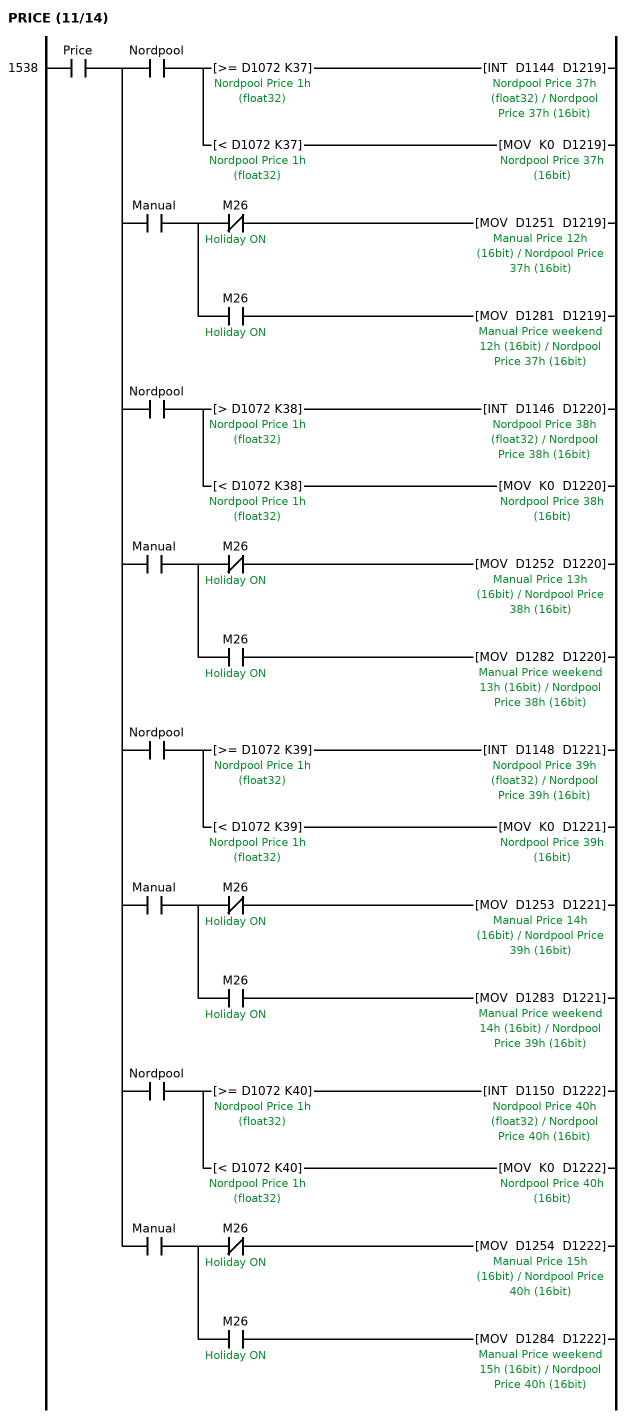
1538  LD      Price
      MPS
      AND     Nordpool
      MPS
      AND>=   D1072 K37  ; Nordpool Price 1h (float32)
      INT     D1144 D1219  ; Nordpool Price 37h (float32) / Nordpool Price 37h (16bit)
        [note] 37-38 (12-13)
      MPP
      AND<    D1072 K37  ; Nordpool Price 1h (float32)
      MOV     K0 D1219
      MRD
      AND     Manual
      MPS
      ANI     M26  ; Holiday ON
      MOV     D1251 D1219
      MPP
      AND     M26  ; Holiday ON
      MOV     D1281 D1219
      MRD
      AND     Nordpool
      MPS
      AND>    D1072 K38  ; Nordpool Price 1h (float32)
      INT     D1146 D1220  ; Nordpool Price 38h (float32) / Nordpool Price 38h (16bit)
        [note] 38-39 (13-14)
      MPP
      AND<    D1072 K38  ; Nordpool Price 1h (float32)
      MOV     K0 D1220
      MRD
      AND     Manual
      MPS
      ANI     M26  ; Holiday ON
      MOV     D1252 D1220
      MPP
      AND     M26  ; Holiday ON
      MOV     D1282 D1220
      MRD
      AND     Nordpool
      MPS
      AND>=   D1072 K39  ; Nordpool Price 1h (float32)
      INT     D1148 D1221  ; Nordpool Price 39h (float32) / Nordpool Price 39h (16bit)
        [note] 39-40 (14-15)
      MPP
      AND<    D1072 K39  ; Nordpool Price 1h (float32)
      MOV     K0 D1221
      MRD
      AND     Manual
      MPS
      ANI     M26  ; Holiday ON
      MOV     D1253 D1221
      MPP
      AND     M26  ; Holiday ON
      MOV     D1283 D1221
      MRD
      AND     Nordpool
      MPS
      AND>=   D1072 K40  ; Nordpool Price 1h (float32)
      INT     D1150 D1222  ; Nordpool Price 40h (float32) / Nordpool Price 40h (16bit)
        [note] 40-41 (15-16)
      MPP
      AND<    D1072 K40  ; Nordpool Price 1h (float32)
      MOV     K0 D1222
      MPP
      AND     Manual
      MPS
      ANI     M26  ; Holiday ON
      MOV     D1254 D1222
      MPP
      AND     M26  ; Holiday ON
      MOV     D1284 D1222
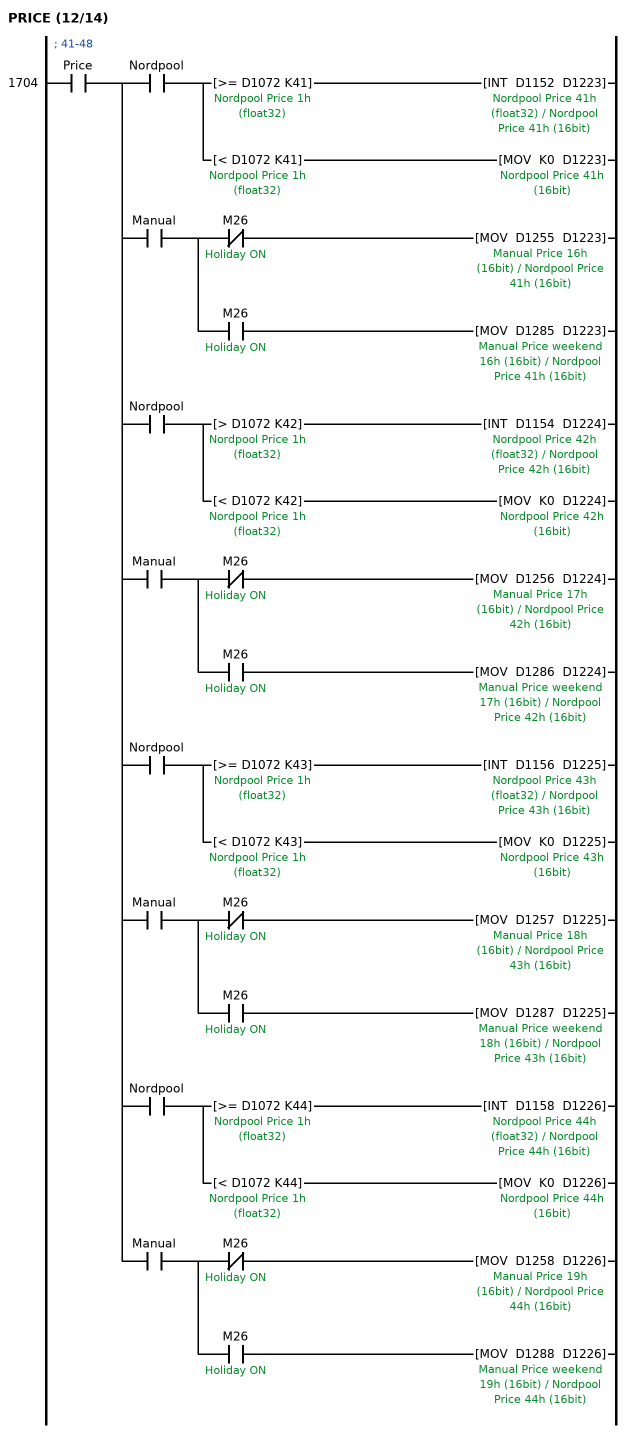
; 41-48
1704  LD      Price
      MPS
      AND     Nordpool
      MPS
      AND>=   D1072 K41  ; Nordpool Price 1h (float32)
      INT     D1152 D1223  ; Nordpool Price 41h (float32) / Nordpool Price 41h (16bit)
        [note] 41-42 (16-17)
      MPP
      AND<    D1072 K41  ; Nordpool Price 1h (float32)
      MOV     K0 D1223
      MRD
      AND     Manual
      MPS
      ANI     M26  ; Holiday ON
      MOV     D1255 D1223
      MPP
      AND     M26  ; Holiday ON
      MOV     D1285 D1223
      MRD
      AND     Nordpool
      MPS
      AND>    D1072 K42  ; Nordpool Price 1h (float32)
      INT     D1154 D1224  ; Nordpool Price 42h (float32) / Nordpool Price 42h (16bit)
        [note] 42-43 (17-18)
      MPP
      AND<    D1072 K42  ; Nordpool Price 1h (float32)
      MOV     K0 D1224
      MRD
      AND     Manual
      MPS
      ANI     M26  ; Holiday ON
      MOV     D1256 D1224
      MPP
      AND     M26  ; Holiday ON
      MOV     D1286 D1224
      MRD
      AND     Nordpool
      MPS
      AND>=   D1072 K43  ; Nordpool Price 1h (float32)
      INT     D1156 D1225  ; Nordpool Price 43h (float32) / Nordpool Price 43h (16bit)
        [note] 43-44 (18-19)
      MPP
      AND<    D1072 K43  ; Nordpool Price 1h (float32)
      MOV     K0 D1225
      MRD
      AND     Manual
      MPS
      ANI     M26  ; Holiday ON
      MOV     D1257 D1225
      MPP
      AND     M26  ; Holiday ON
      MOV     D1287 D1225
      MRD
      AND     Nordpool
      MPS
      AND>=   D1072 K44  ; Nordpool Price 1h (float32)
      INT     D1158 D1226  ; Nordpool Price 44h (float32) / Nordpool Price 44h (16bit)
        [note] 44-45 (19-20)
      MPP
      AND<    D1072 K44  ; Nordpool Price 1h (float32)
      MOV     K0 D1226
      MPP
      AND     Manual
      MPS
      ANI     M26  ; Holiday ON
      MOV     D1258 D1226
      MPP
      AND     M26  ; Holiday ON
      MOV     D1288 D1226
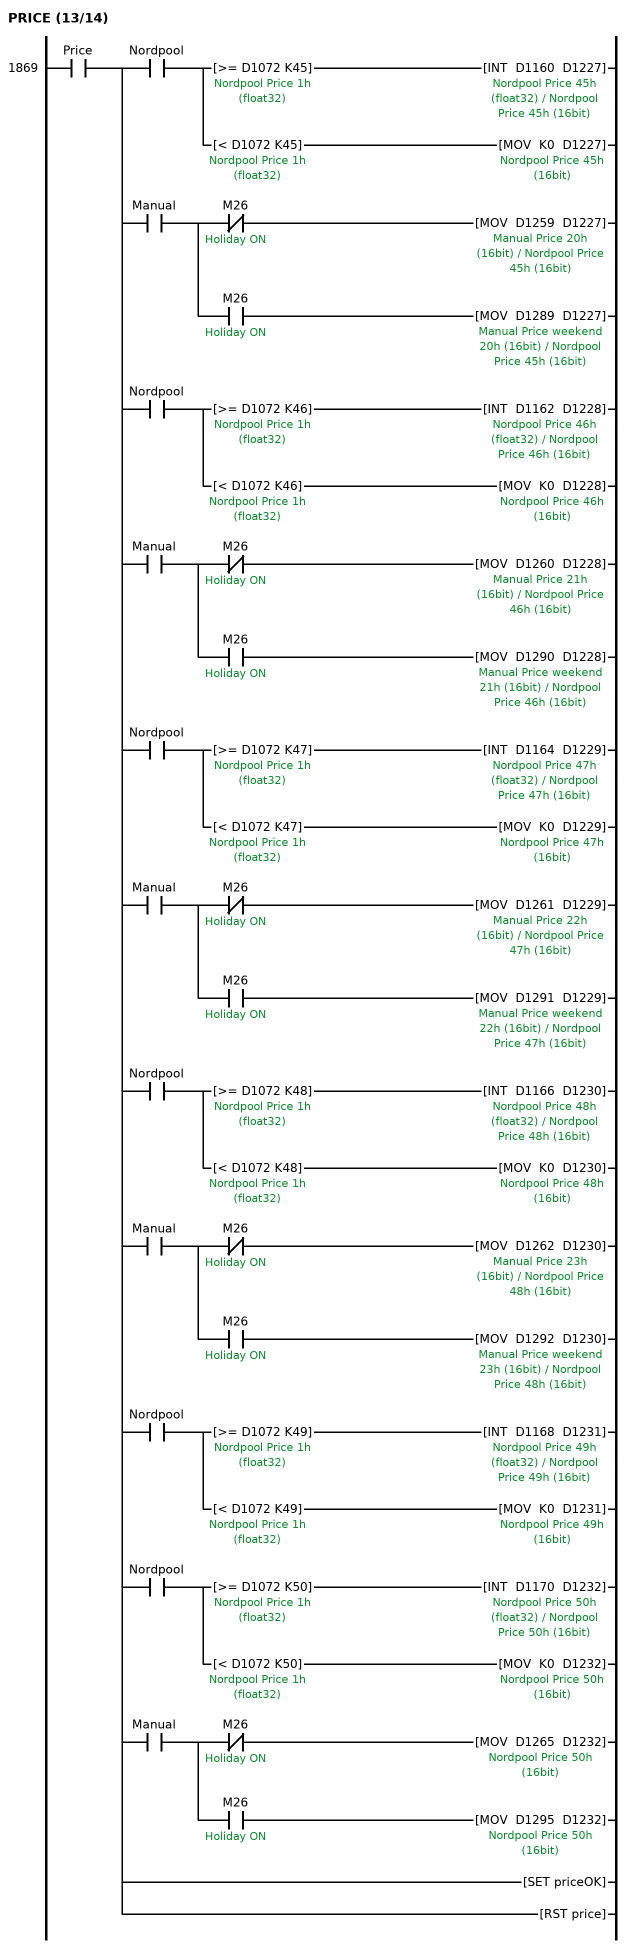
1869  LD      Price
      MPS
      AND     Nordpool
      MPS
      AND>=   D1072 K45  ; Nordpool Price 1h (float32)
      INT     D1160 D1227  ; Nordpool Price 45h (float32) / Nordpool Price 45h (16bit)
        [note] 45-46 (20-21)
      MPP
      AND<    D1072 K45  ; Nordpool Price 1h (float32)
      MOV     K0 D1227
      MRD
      AND     Manual
      MPS
      ANI     M26  ; Holiday ON
      MOV     D1259 D1227
      MPP
      AND     M26  ; Holiday ON
      MOV     D1289 D1227
      MRD
      AND     Nordpool
      MPS
      AND>=   D1072 K46  ; Nordpool Price 1h (float32)
      INT     D1162 D1228  ; Nordpool Price 46h (float32) / Nordpool Price 46h (16bit)
        [note] 46-47 (21-22)
      MPP
      AND<    D1072 K46  ; Nordpool Price 1h (float32)
      MOV     K0 D1228
      MRD
      AND     Manual
      MPS
      ANI     M26  ; Holiday ON
      MOV     D1260 D1228
      MPP
      AND     M26  ; Holiday ON
      MOV     D1290 D1228
      MRD
      AND     Nordpool
      MPS
      AND>=   D1072 K47  ; Nordpool Price 1h (float32)
      INT     D1164 D1229  ; Nordpool Price 47h (float32) / Nordpool Price 47h (16bit)
        [note] 47-48 (22-23)
      MPP
      AND<    D1072 K47  ; Nordpool Price 1h (float32)
      MOV     K0 D1229
      MRD
      AND     Manual
      MPS
      ANI     M26  ; Holiday ON
      MOV     D1261 D1229
      MPP
      AND     M26  ; Holiday ON
      MOV     D1291 D1229
      MRD
      AND     Nordpool
      MPS
      AND>=   D1072 K48  ; Nordpool Price 1h (float32)
      INT     D1166 D1230  ; Nordpool Price 48h (float32) / Nordpool Price 48h (16bit)
        [note] 48-49 (23-24)
      MPP
      AND<    D1072 K48  ; Nordpool Price 1h (float32)
      MOV     K0 D1230
      MRD
      AND     Manual
      MPS
      ANI     M26  ; Holiday ON
      MOV     D1262 D1230
      MPP
      AND     M26  ; Holiday ON
      MOV     D1292 D1230
      MRD
      AND     Nordpool
      MPS
      AND>=   D1072 K49  ; Nordpool Price 1h (float32)
      INT     D1168 D1231  ; Nordpool Price 49h (float32) / Nordpool Price 49h (16bit)
        [note] 49-50 (00-01)
      MPP
      AND<    D1072 K49  ; Nordpool Price 1h (float32)
      MOV     K0 D1231
      MRD
      AND     Nordpool
      MPS
      AND>=   D1072 K50  ; Nordpool Price 1h (float32)
      INT     D1170 D1232  ; Nordpool Price 50h (float32) / Nordpool Price 50h (16bit)
      MPP
      AND<    D1072 K50  ; Nordpool Price 1h (float32)
      MOV     K0 D1232
      MRD
      AND     Manual
      MPS
      ANI     M26  ; Holiday ON
      MOV     D1265 D1232
      MPP
      AND     M26  ; Holiday ON
      MOV     D1295 D1232
      MPP
      SET     priceOK
      RST     price
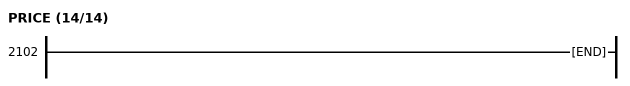
2102  END
END_PROGRAM

PROGRAM 15_00_UP
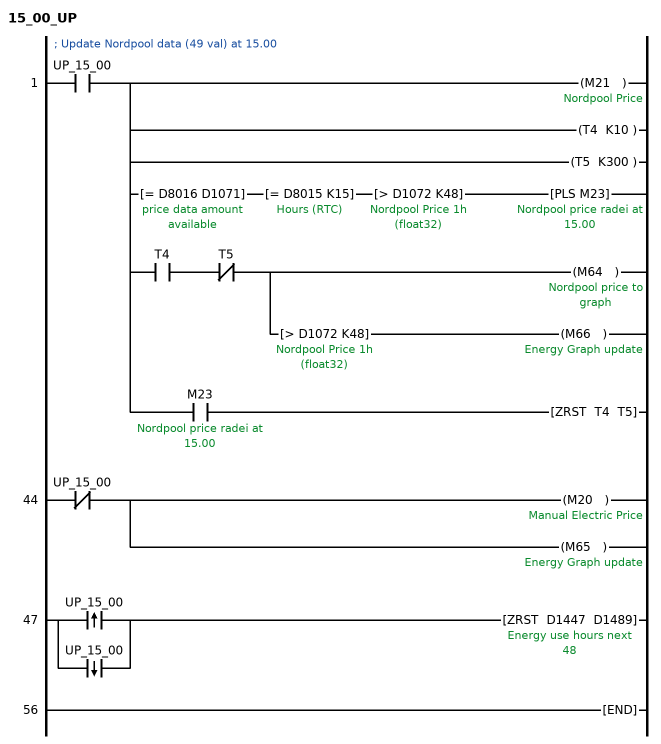
; Update Nordpool data (49 val) at 15.00
1     LD      UP_15_00
      OUT     M21  ; Nordpool Price
      OUT     T4 K10
      OUT     T5 K300
      MPS
      AND=    D8016 D1071  ; price data amount available
      AND=    D8015 K15  ; Hours (RTC)
      AND>    D1072 K48  ; Nordpool Price 1h (float32)
      PLS     M23  ; Nordpool price radei at 15.00
      MRD
      AND     T4
      ANI     T5
      OUT     M64  ; Nordpool price to graph
      AND>    D1072 K48  ; Nordpool Price 1h (float32)
      OUT     M66  ; Energy Graph update
      MPP
      AND     M23  ; Nordpool price radei at 15.00
      ZRST    T4 T5
44    LDI     UP_15_00
      OUT     M20  ; Manual Electric Price
      OUT     M65  ; Energy Graph update
47    LDP     UP_15_00
      ORF     UP_15_00
      ZRST    D1447 D1489  ; Energy use hours next 48
56    END
END_PROGRAM

PROGRAM Hour_Use
VAR
  EnernyUse : BOOL;  (* Select good time *)
END_VAR
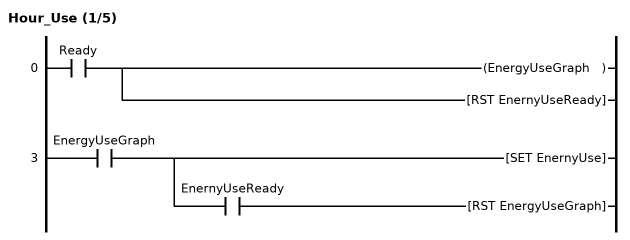
0     LD      Ready
      OUT     EnergyUseGraph
      RST     EnernyUseReady
3     LD      EnergyUseGraph
      SET     EnernyUse
      AND     EnernyUseReady
      RST     EnergyUseGraph
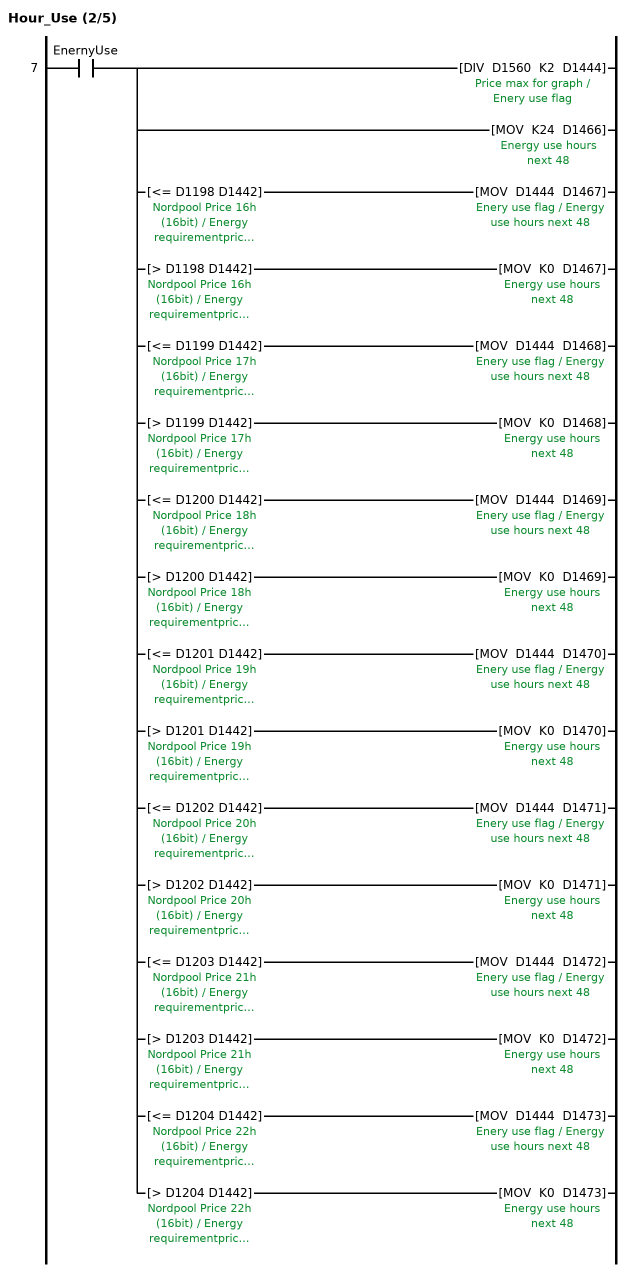
7     LD      EnernyUse
      DIV     D1560 K2 D1444  ; Price max for graph / Enery use flag
        [note] 15.00
      MOV     K24 D1466  ; Energy use hours next 48
      MPS
      AND<=   D1198 D1442  ; Nordpool Price 16h (16bit) / Energy requirementprice level
      MOV     D1444 D1467  ; Energy use hours next 48
      MRD
      AND>    D1198 D1442  ; Nordpool Price 16h (16bit) / Energy requirementprice level
      MOV     K0 D1467
      MRD
      AND<=   D1199 D1442  ; Nordpool Price 17h (16bit) / Energy requirementprice level
      MOV     D1444 D1468  ; Energy use hours next 48
        [note] 16.00
      MRD
      AND>    D1199 D1442  ; Nordpool Price 17h (16bit) / Energy requirementprice level
      MOV     K0 D1468
      MRD
      AND<=   D1200 D1442  ; Nordpool Price 18h (16bit) / Energy requirementprice level
      MOV     D1444 D1469  ; Energy use hours next 48
        [note] 17.00
      MRD
      AND>    D1200 D1442  ; Nordpool Price 18h (16bit) / Energy requirementprice level
      MOV     K0 D1469
      MRD
      AND<=   D1201 D1442  ; Nordpool Price 19h (16bit) / Energy requirementprice level
      MOV     D1444 D1470  ; Energy use hours next 48
        [note] 18.00
      MRD
      AND>    D1201 D1442  ; Nordpool Price 19h (16bit) / Energy requirementprice level
      MOV     K0 D1470
      MRD
      AND<=   D1202 D1442  ; Nordpool Price 20h (16bit) / Energy requirementprice level
      MOV     D1444 D1471  ; Energy use hours next 48
        [note] 19.00
      MRD
      AND>    D1202 D1442  ; Nordpool Price 20h (16bit) / Energy requirementprice level
      MOV     K0 D1471
      MRD
      AND<=   D1203 D1442  ; Nordpool Price 21h (16bit) / Energy requirementprice level
      MOV     D1444 D1472  ; Energy use hours next 48
        [note] 20.00
      MRD
      AND>    D1203 D1442  ; Nordpool Price 21h (16bit) / Energy requirementprice level
      MOV     K0 D1472
      MRD
      AND<=   D1204 D1442  ; Nordpool Price 22h (16bit) / Energy requirementprice level
      MOV     D1444 D1473  ; Energy use hours next 48
        [note] 21.00
      MPP
      AND>    D1204 D1442  ; Nordpool Price 22h (16bit) / Energy requirementprice level
      MOV     K0 D1473
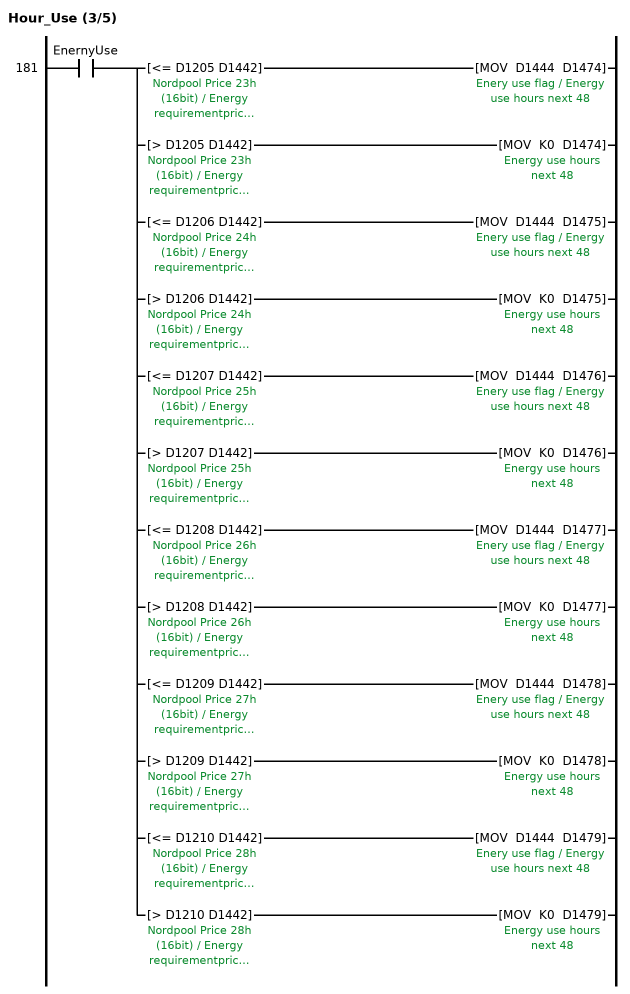
181   LD      EnernyUse
      MPS
      AND<=   D1205 D1442  ; Nordpool Price 23h (16bit) / Energy requirementprice level
      MOV     D1444 D1474  ; Energy use hours next 48
        [note] 22.00
      MRD
      AND>    D1205 D1442  ; Nordpool Price 23h (16bit) / Energy requirementprice level
      MOV     K0 D1474
      MRD
      AND<=   D1206 D1442  ; Nordpool Price 24h (16bit) / Energy requirementprice level
      MOV     D1444 D1475  ; Energy use hours next 48
        [note] 23.00
      MRD
      AND>    D1206 D1442  ; Nordpool Price 24h (16bit) / Energy requirementprice level
      MOV     K0 D1475
      MRD
      AND<=   D1207 D1442  ; Nordpool Price 25h (16bit) / Energy requirementprice level
      MOV     D1444 D1476  ; Energy use hours next 48
        [note] 24.00 (24-01)
      MRD
      AND>    D1207 D1442  ; Nordpool Price 25h (16bit) / Energy requirementprice level
      MOV     K0 D1476
      MRD
      AND<=   D1208 D1442  ; Nordpool Price 26h (16bit) / Energy requirementprice level
      MOV     D1444 D1477  ; Energy use hours next 48
        [note] 25.00 01-02
      MRD
      AND>    D1208 D1442  ; Nordpool Price 26h (16bit) / Energy requirementprice level
      MOV     K0 D1477
      MRD
      AND<=   D1209 D1442  ; Nordpool Price 27h (16bit) / Energy requirementprice level
      MOV     D1444 D1478  ; Energy use hours next 48
        [note] 26.00 02-03
      MRD
      AND>    D1209 D1442  ; Nordpool Price 27h (16bit) / Energy requirementprice level
      MOV     K0 D1478
      MRD
      AND<=   D1210 D1442  ; Nordpool Price 28h (16bit) / Energy requirementprice level
      MOV     D1444 D1479  ; Energy use hours next 48
        [note] 27.00 03-04
      MPP
      AND>    D1210 D1442  ; Nordpool Price 28h (16bit) / Energy requirementprice level
      MOV     K0 D1479
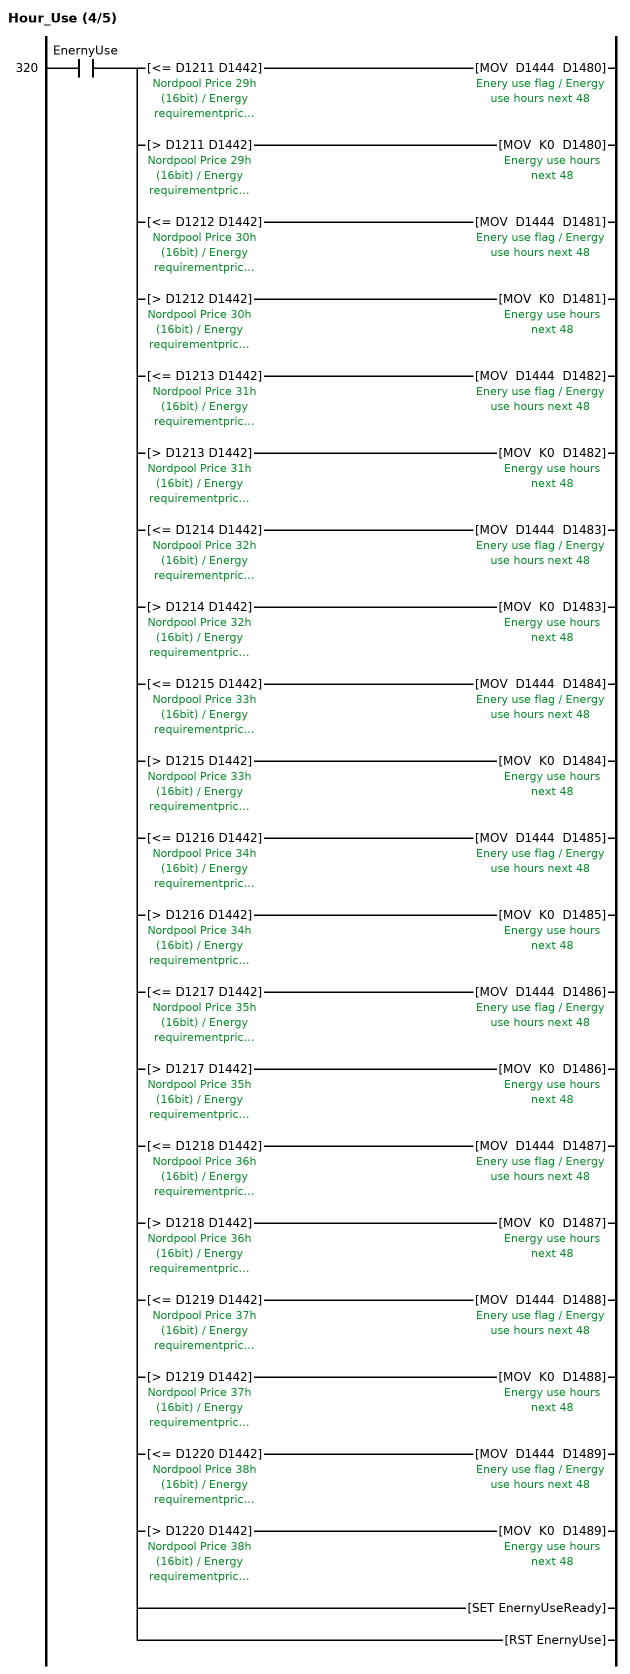
320   LD      EnernyUse
      MPS
      AND<=   D1211 D1442  ; Nordpool Price 29h (16bit) / Energy requirementprice level
      MOV     D1444 D1480  ; Energy use hours next 48
        [note] 28.00 04-05
      MRD
      AND>    D1211 D1442  ; Nordpool Price 29h (16bit) / Energy requirementprice level
      MOV     K0 D1480
      MRD
      AND<=   D1212 D1442  ; Nordpool Price 30h (16bit) / Energy requirementprice level
      MOV     D1444 D1481  ; Energy use hours next 48
        [note] 29.00 05-06
      MRD
      AND>    D1212 D1442  ; Nordpool Price 30h (16bit) / Energy requirementprice level
      MOV     K0 D1481
      MRD
      AND<=   D1213 D1442  ; Nordpool Price 31h (16bit) / Energy requirementprice level
      MOV     D1444 D1482  ; Energy use hours next 48
        [note] 30.00 06-07
      MRD
      AND>    D1213 D1442  ; Nordpool Price 31h (16bit) / Energy requirementprice level
      MOV     K0 D1482
      MRD
      AND<=   D1214 D1442  ; Nordpool Price 32h (16bit) / Energy requirementprice level
      MOV     D1444 D1483  ; Energy use hours next 48
        [note] 31.00 07-08
      MRD
      AND>    D1214 D1442  ; Nordpool Price 32h (16bit) / Energy requirementprice level
      MOV     K0 D1483
      MRD
      AND<=   D1215 D1442  ; Nordpool Price 33h (16bit) / Energy requirementprice level
      MOV     D1444 D1484  ; Energy use hours next 48
        [note] 32.00 08-09
      MRD
      AND>    D1215 D1442  ; Nordpool Price 33h (16bit) / Energy requirementprice level
      MOV     K0 D1484
      MRD
      AND<=   D1216 D1442  ; Nordpool Price 34h (16bit) / Energy requirementprice level
      MOV     D1444 D1485  ; Energy use hours next 48
        [note] 33.00 09-10
      MRD
      AND>    D1216 D1442  ; Nordpool Price 34h (16bit) / Energy requirementprice level
      MOV     K0 D1485
      MRD
      AND<=   D1217 D1442  ; Nordpool Price 35h (16bit) / Energy requirementprice level
      MOV     D1444 D1486  ; Energy use hours next 48
        [note] 34.00 10-11
      MRD
      AND>    D1217 D1442  ; Nordpool Price 35h (16bit) / Energy requirementprice level
      MOV     K0 D1486
      MRD
      AND<=   D1218 D1442  ; Nordpool Price 36h (16bit) / Energy requirementprice level
      MOV     D1444 D1487  ; Energy use hours next 48
        [note] 35.00 11-12
      MRD
      AND>    D1218 D1442  ; Nordpool Price 36h (16bit) / Energy requirementprice level
      MOV     K0 D1487
      MRD
      AND<=   D1219 D1442  ; Nordpool Price 37h (16bit) / Energy requirementprice level
      MOV     D1444 D1488  ; Energy use hours next 48
        [note] 36.00 12-13
      MRD
      AND>    D1219 D1442  ; Nordpool Price 37h (16bit) / Energy requirementprice level
      MOV     K0 D1488
      MRD
      AND<=   D1220 D1442  ; Nordpool Price 38h (16bit) / Energy requirementprice level
      MOV     D1444 D1489  ; Energy use hours next 48
        [note] 36.00 13-14
      MRD
      AND>    D1220 D1442  ; Nordpool Price 38h (16bit) / Energy requirementprice level
      MOV     K0 D1489
      MPP
      SET     EnernyUseReady
      RST     EnernyUse
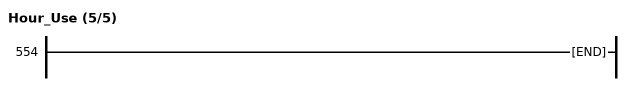
554   END
END_PROGRAM

PROGRAM PtoGaph
VAR
  DataCopy : BOOL;  (* Data copy *)
END_VAR
